// POUs/Diverse/FB_SafetyElementAnz
// Dieser FB dient zur Erweiterung eines älteren Schutztürbausteins für die Anzeige (nur Anzeige keine Fehlermeldung) in der Avalon-HMI im DataCrtlView oder PlcStructure.
// Zudem kann er noch als AnzeigeFB für Lichtgitter oder einzelne Nothalte genuzt werden.
FUNCTION_BLOCK FB_SafetyElementAnz
VAR_IN_OUT
	IQ_stOpVisual			:ST_OP_Visual;	// Zur Anzeige der Schutztür mit Nothalt oder auch Lichtgitter in der HMI
END_VAR
VAR_INPUT
	I_bTuerGeschlossen	: BOOL	:= TRUE;	// Türschalter: TwinSAFE-Kanal 1 geschlossen, oder Lichtgitter OK, oder wenn nur der Nothalt zur Anzeige gebracht wird, weglassen
	I_bTuerGeschlUndVerr	: BOOL	:= TRUE;	// Türschalter: TwinSAFE-Kanal 2 verriegelt, oder Lichtgitter OK, oder wenn nur der Nothalt zur Anzeige gebracht wird, weglassen
	I_bAutoHalt				: BOOL;	// Autohalt der Schutztür aktiv
	I_bNotHalt				: BOOL	:= TRUE;	//	Nothalt an der Schutztür wurde gedrückt, bei Lichtgitter einfach weglassen
	I_bTakt					: BOOL;	//  blinktakt für Q_bAnzeige
	I_sPfadImage			: STRING	:='Objekt-Schiebetuer.svg';	//Pfad für das anzuzeigende Icon
END_VAR
VAR_OUTPUT
	Q_nAnzeige				: DWORD;	// Für die Anzeige im DataCrtlView: Farbe, rot bei Nothalt, gelb bei offen und blau bei Automatik-Halt
	Q_bAnzeige				: BOOL;	// Für die Anzeige im DataCrtlView: TRUE bei Nothalt oder wenn die Tür nicht geschlossen und verriegelt ist
END_VAR

IQ_stOpVisual.sImage := I_sPfadImage;

IF NOT I_bNotHalt
THEN
	IQ_stOpVisual.sColour := cRotAsString;
	IQ_stOpVisual.iDisplayMode := 1;
	Q_bAnzeige	:= TRUE;
	IF I_bTakt
	THEN
		Q_nAnzeige	:= cRot;
	ELSE
		Q_nAnzeige	:= cKEYBACK;
	END_IF
ELSIF I_bTuerGeschlossen
	AND I_bTuerGeschlUndVerr
	AND I_bAutoHalt
THEN
	IQ_stOpVisual.iDisplayMode := 1;
	IQ_stOpVisual.sColour := cBlauAsString;
ELSIF I_bTuerGeschlossen
	AND I_bTuerGeschlUndVerr
THEN
	IQ_stOpVisual.sColour := cDefaultAsString;
	Q_bAnzeige	:= FALSE;
	Q_nAnzeige	:= cKEYBACK;
	IQ_stOpVisual.iDisplayMode := 3;
ELSE
	IQ_stOpVisual.sColour := cGelbAsString;
	IQ_stOpVisual.iDisplayMode := 1;
	Q_bAnzeige	:= TRUE;
	IF I_bTakt
	THEN
		Q_nAnzeige	:= cGelb;
	ELSE
		Q_nAnzeige	:= cKEYBACK;
	END_IF
END_IF

END_FUNCTION_BLOCK

// POUs/Diverse/FB_UsvStatus
// Dieser Baustein wertet die lokale USV aus und beschreibt die Meldungen.
// Es ist eigentlich nur eine Übersetzung von dem USV-Baustein auf die Avalon-Meldungen
FUNCTION_BLOCK FB_UsvStatus
VAR_INPUT
	I_nLevelLowPercent		:	DWORD:= 30;
	I_nLevelCriticalPercent	:	DWORD:= 15;
END_VAR
VAR_IN_OUT
	IQ_stMeldung			: ST_MeldUSV;
END_VAR
VAR
	fbGetUPSStatus		:	Tc2_IoFunctions.FB_GetUPSStatus;
END_VAR

fbGetUPSStatus(
	sNetId		:=	'',
	nPort			:=	0,		// 0 = Windows UPS service
	bEnable		:=	TRUE
);

IQ_stMeldung.bMeldAustausch			:= fbGetUPSStatus.stStatus.eBatteryStatus	=	Tc2_IoFunctions.BatteryReplace;
IQ_stMeldung.bMeldBatteriebetrieb	:= fbGetUPSStatus.stStatus.ePowerStatus	=	Tc2_IoFunctions.PowerOnBattery;
IQ_stMeldung.bMeldKommFehler			:= fbGetUPSStatus.stStatus.eCommStatus	=	Tc2_IoFunctions.UpsCommFailed;
IQ_stMeldung.bMeldKritLevel			:= fbGetUPSStatus.stStatus.BatteryLifePercent < I_nLevelCriticalPercent;
IQ_stMeldung.bMeldStatusUnbekannt	:= fbGetUPSStatus.stStatus.eCommStatus	=	Tc2_IoFunctions.UpsCommUnknownStatus;
IQ_stMeldung.bMeldUnteresLevel		:= fbGetUPSStatus.stStatus.BatteryLifePercent < I_nLevelLowPercent
													AND fbGetUPSStatus.stStatus.ePowerStatus	=	Tc2_IoFunctions.PowerOnBattery;
// ENDE

END_FUNCTION_BLOCK

// POUs/Diverse/FB_WartgTuer
// OBSOLET! Wird nicht weiter supportet. FB für eine Wartungstür. Noch keine Adaption an die Avalon-HMI.
// Es sollte der FB_WartgTuerMeld genutzt werden.
FUNCTION_BLOCK FB_WartgTuer
VAR_INPUT
	I_bFreigTuerEntrieg	:BOOL;	//Allgem. Türfreigabe durch PLC
	I_bAnAbwTastEntrieg	:BOOL;
	I_bQuittTastVerrieg	:BOOL;
	I_bAbfrgTuerGeschl	:BOOL;	//Türschalter: TwinSAFE-Kanal 1
	I_bAbfrgTuerMagnet	:BOOL;	//Türschalter: TwinSAFE-Kanal 2	
	I_bEntrgMeldMagnet	:BOOL;	//Rückmeldung vom Safety-Projekt
	I_bHinwTaktEntrieg	:BOOL;
	I_bHinwTaktEntrglt	:BOOL;

	I_bAutomBetrAngew		:BOOL;
	I_bTastAutomForts		:BOOL;
	I_bUeberbrSteuerhilfsluft	: BOOL;
END_VAR
VAR_OUTPUT

	Q_bAnwTuerEntrieg		:BOOL; 
	Q_bTuerEntriegelt		:BOOL; 
	Q_bAnwQuittMeldg		:BOOL; 
	Q_bEntrgAnfdMagnet	:BOOL;	//Anforderung an Safety-Projekt

	Q_bAutomHaltAktiv		:BOOL;
	Q_bAutomHaltMeldg		:BOOL;	
	
	Q_bAutomHaltMeldgHin	:BOOL;
	
END_VAR
VAR

	
	rtrigAnwQuittTast		:R_TRIG;
	bAnwahlEntriegeln		:BOOL;
	bMagnetEntriegeln		:BOOL;
	bMagnetEntriegelt		:BOOL;
	
	rtrigTastAutoForts	:R_TRIG;
	bAutomHaltManForts	:BOOL;
	
	tonInit					:TON;
	
END_VAR

a_TuerEntrieg ();
b_AutomHalt ();

ACTION a_TuerEntrieg:

//Init, da die Signale aus der Safety nicht sofort da sind und dann die Türen sich öffnen	
tonInit(	IN:= TRUE,
			PT:= T#5S);	
	
IF tonInit.Q
	AND bTwinSAFEInRun
THEN

	rtrigAnwQuittTast (CLK:= I_bAnAbwTastEntrieg
							  		 OR I_bQuittTastVerrieg); 
	
	IF I_bAnAbwTastEntrieg
		AND rtrigAnwQuittTast.Q
		AND NOT bMagnetEntriegelt
	THEN
		bAnwahlEntriegeln:= NOT bAnwahlEntriegeln;	
	END_IF
	
	IF (I_bQuittTastVerrieg
		AND rtrigAnwQuittTast.Q)	
		AND I_bAbfrgTuerGeschl
	THEN
		bMagnetEntriegeln:=	
		bMagnetEntriegelt:= FALSE;	
	END_IF	

	IF (bAnwahlEntriegeln
			AND I_bFreigTuerEntrieg)
		OR NOT I_bAbfrgTuerGeschl
		OR (NOT I_bQuittTastVerrieg
				AND NOT I_bAbfrgTuerMagnet) 
	THEN
		bMagnetEntriegeln:= TRUE;		

		IF I_bEntrgMeldMagnet 
		THEN
			bAnwahlEntriegeln:= FALSE;
			bMagnetEntriegelt:= TRUE;	
		END_IF
   END_IF

	(*Ausgangszuweisung*)

	Q_bAnwTuerEntrieg := bAnwahlEntriegeln;
	
	Q_bTuerEntriegelt	:= bMagnetEntriegelt;
	
	Q_bAnwQuittMeldg	:= (bAnwahlEntriegeln
									AND I_bHinwTaktEntrieg) 
								OR ((NOT I_bAbfrgTuerGeschl
										OR NOT I_bAbfrgTuerMagnet)
									AND I_bHinwTaktEntrglt)
								OR (NOT bAnwahlEntriegeln
										AND NOT bMagnetEntriegeln);	 

	Q_bEntrgAnfdMagnet:= bMagnetEntriegeln;		
END_IF
END_ACTION

ACTION b_AutomHalt:
	(*Abfrage/Quittierung*)

	rtrigTastAutoForts (CLK:= I_bTastAutomForts
										AND NOT I_bAnAbwTastEntrieg );
	
	IF I_bAutomBetrAngew
		AND bMagnetEntriegelt
	THEN
		bAutomHaltManForts:= TRUE;	
	ELSIF rtrigTastAutoForts.Q 
	THEN
			bAutomHaltManForts:= FALSE;	
   END_IF

	(*Ausgangszuweisung*)

	Q_bAutomHaltAktiv	:= bAutomHaltManForts;
	
	Q_bAutomHaltMeldg	:= (NOT bMagnetEntriegelt
									AND bAutomHaltManForts
									AND I_bHinwTaktEntrglt)
								OR (I_bUeberbrSteuerhilfsluft
										AND (bAnwahlEntriegeln
												OR bMagnetEntriegelt)
									AND NOT I_bHinwTaktEntrglt);
								
	Q_bAutomHaltMeldgHin := NOT bMagnetEntriegelt
									AND bAutomHaltManForts;
END_ACTION

END_FUNCTION_BLOCK

// POUs/Diverse/FB_WartgTuerMeld
// FB für eine Wartungstür mit einem Taster zum Umschalten der Schutztüranforderung/Quittierung und einem Taster für Automatikablauf starten.
// Dieser FB ist für die Verwendung mit der Avalon-HMI vorgesehen.
FUNCTION_BLOCK FB_WartgTuerMeld
VAR_IN_OUT		
	IQ_stMeldHMI			:ST_MeldWartgTuer;	// HMI-Strukturen
END_VAR
VAR_INPUT
	I_sName					:STRING;	// Name der Schutztür
	I_sBMK					:STRING;	// z.B.:"ST1020"
	I_bFreigTuerEntrieg	:BOOL;	// Allgem. Türfreigabe durch PLC
	I_bAnAbwTastEntrieg	:BOOL;	// Hardwaretaste für Schutztür anfordern/quittieren
	I_bQuittTastVerrieg	:BOOL;	// Hardwaretaste für Schutztür anfordern/quittieren
	I_bAbfrgTuerGeschl	:BOOL;	// Türschalter: TwinSAFE-Kanal 1
	I_bAbfrgTuerMagnet	:BOOL;	// Türschalter: TwinSAFE-Kanal 2	
	I_bEntrgMeldMagnet	:BOOL;	// Rückmeldung vom Safety-Projekt
	I_bHinwTaktEntrieg	:BOOL;	// mittlerer Takt, ggf. 1Hz
	I_bHinwTaktEntrglt	:BOOL;	// schneller Takt, ggf. 5Hz

	I_bAutomBetrAngew		:BOOL;	// Signal das Automatikablauf angewählt ist.
	I_bTastAutomForts		:BOOL;	// Hardwaretaste für Automatikablauf fortsetzen
	I_bUeberbrSteuerhilfsluft	: BOOL;	// Signal aus dem Safety: Steuerhilfluft ist überbrückt
	
	I_bMeldFreigabe		:BOOL	:= TRUE;	// Hiermit wird die Meldung in der HMI freigegeben. Dieser Eingang kann mit TwinSAFE_OK (oder ähnliches) beschrieben werden, damit die Meldung bei einem Safetyfehler nicht angezeigt werden und unnötig die Meldungen zumüllen.
END_VAR
VAR_OUTPUT

	Q_bAnwTuerEntrieg		:BOOL; 	// Meldung Wartungstür ist zum Entriegeln angwählt
	Q_bTuerEntriegelt		:BOOL;	// Meldung Wartungstür ist entriegelt
	Q_bAnwQuittMeldg		:BOOL;	// Leuchtmelder für den Taster Schutztür anfordern/quittieren
	Q_bEntrgAnfdMagnet	:BOOL;	// Anforderung an Safety-Projekt

	Q_bAutomHaltAktiv		:BOOL;	// Meldung Automatik-Halt ist aktiv
	Q_bAutomHaltMeldg		:BOOL;	// Leuchtmelder für den Taster Automatikablauf fortsetzen
	
	Q_bAutomHaltMeldgHin	:BOOL;	// Meldung das Automatik-Halt noch aktiv ist, obwohl Schutztür geschlossen ist.
	
END_VAR
VAR

	
	rtrigAnwQuittTast		:R_TRIG;
	bAnwahlEntriegeln		:BOOL;
	bMagnetEntriegeln		:BOOL;
	bMagnetEntriegelt		:BOOL;
	
	rtrigTastAutoForts	:R_TRIG;
	bAutomHaltManForts	:BOOL;
	
	tonInit					:TON;
	
END_VAR

a_TuerEntrieg ();
b_AutomHalt ();
z_Meld();

ACTION a_TuerEntrieg:

//Init, da die Signale aus der Safety nicht sofort da sind und dann die Türen sich öffnen	
tonInit(	IN:= TRUE,
			PT:= T#5S);	
	
IF tonInit.Q
	AND bTwinSAFEInRun
THEN

	rtrigAnwQuittTast (CLK:= I_bAnAbwTastEntrieg
							  		 OR I_bQuittTastVerrieg); 
	
	IF I_bAnAbwTastEntrieg
		AND rtrigAnwQuittTast.Q
		AND NOT bMagnetEntriegelt
	THEN
		bAnwahlEntriegeln:= NOT bAnwahlEntriegeln;	
	END_IF
	
	IF (I_bQuittTastVerrieg
		AND rtrigAnwQuittTast.Q)	
		AND I_bAbfrgTuerGeschl
	THEN
		bMagnetEntriegeln:=	
		bMagnetEntriegelt:= FALSE;	
	END_IF	

	IF (bAnwahlEntriegeln
			AND I_bFreigTuerEntrieg)
		OR NOT I_bAbfrgTuerGeschl
		OR (NOT I_bQuittTastVerrieg
				AND NOT I_bAbfrgTuerMagnet) 
	THEN
		bMagnetEntriegeln:= TRUE;		

		IF I_bEntrgMeldMagnet 
		THEN
			bAnwahlEntriegeln:= FALSE;
			bMagnetEntriegelt:= TRUE;	
		END_IF
   END_IF

	(*Ausgangszuweisung*)

	Q_bAnwTuerEntrieg := bAnwahlEntriegeln;
	
	Q_bTuerEntriegelt	:= bMagnetEntriegelt;
	
	Q_bAnwQuittMeldg	:= (bAnwahlEntriegeln
									AND I_bHinwTaktEntrieg) 
								OR ((NOT I_bAbfrgTuerGeschl
										OR NOT I_bAbfrgTuerMagnet)
									AND I_bHinwTaktEntrglt)
								OR (NOT bAnwahlEntriegeln
									AND NOT bMagnetEntriegeln);	 

	Q_bEntrgAnfdMagnet:= bMagnetEntriegeln;		
END_IF
END_ACTION

ACTION b_AutomHalt:
	(*Abfrage/Quittierung*)

	rtrigTastAutoForts (CLK:= I_bTastAutomForts
										AND NOT I_bAnAbwTastEntrieg );
	
	IF I_bAutomBetrAngew
		AND bMagnetEntriegelt
	THEN
		bAutomHaltManForts:= TRUE;	
	ELSIF rtrigTastAutoForts.Q 
	THEN
			bAutomHaltManForts:= FALSE;	
   END_IF

	(*Ausgangszuweisung*)

	Q_bAutomHaltAktiv	:= bAutomHaltManForts;
	
	Q_bAutomHaltMeldg	:= (NOT bMagnetEntriegelt
									AND bAutomHaltManForts
									AND I_bHinwTaktEntrglt)
								OR (I_bUeberbrSteuerhilfsluft
										AND (bAnwahlEntriegeln
												OR bMagnetEntriegelt)
									AND NOT I_bHinwTaktEntrglt);
								
	Q_bAutomHaltMeldgHin := NOT bMagnetEntriegelt
									AND bAutomHaltManForts;
END_ACTION

ACTION z_Meld:


IQ_stMeldHMI.SourceName		 	:= 'Schutztür';
IQ_stMeldHMI.sBMK		 			:= I_sBMK;
IQ_stMeldHMI.sAktorName		 	:= I_sName;
IQ_stMeldHMI.bMeldAutoHalt 	:= Q_bAutomHaltAktiv
											AND NOT Q_bTuerEntriegelt;
											
IQ_stMeldHMI.bMeldGeoeffnet 	:= (NOT I_bAbfrgTuerGeschl
												OR NOT I_bAbfrgTuerMagnet)
											AND I_bMeldFreigabe;
											
IQ_stMeldHMI.bMeldAnwahl		:= bAnwahlEntriegeln
											AND I_bAbfrgTuerMagnet;
END_ACTION

END_FUNCTION_BLOCK

// POUs/Diverse/FB_WartgTuerMeldAnz
// FB für eine Wartungstür mit einem Taster zum Umschalten der Schutztüranforderung/Quittierung und einem Taster für Automatikablauf starten.
// Dieser FB ist für die Verwendung mit der Avalon-HMI vorgesehen und wurde durch eine Anzeigemöglichkeit mit ST_OP_Visual in der Avalon-HMI erweitert.
FUNCTION_BLOCK FB_WartgTuerMeldAnz
VAR_IN_OUT		
	IQ_stMeldHMI			:ST_MeldWartgTuer;	// HMI-Strukturen
	IQ_stOpVisual			:ST_OP_Visual;	// Zur Anzeige der Schutztür mit Nothalt in der HMI
END_VAR
VAR_INPUT
	I_sName					:STRING;	// Name der Schutztür
	I_sBMK					:STRING;	// z.B.:"ST1020"
	I_bFreigTuerEntrieg	:BOOL;	// Allgem. Türfreigabe durch PLC
	I_bAnAbwTastEntrieg	:BOOL;	// Hardwaretaste für Schutztür anfordern/quittieren
	I_bQuittTastVerrieg	:BOOL;	// Hardwaretaste für Schutztür anfordern/quittieren
	I_bAbfrgTuerGeschl	:BOOL;	// Türschalter: TwinSAFE-Kanal 1
	I_bAbfrgTuerMagnet	:BOOL;	// Türschalter: TwinSAFE-Kanal 2	
	I_bEntrgMeldMagnet	:BOOL;	// Rückmeldung vom Safety-Projekt
	I_bHinwTaktEntrieg	:BOOL;	// mittlerer Takt, ggf. 1Hz
	I_bHinwTaktEntrglt	:BOOL;	// schneller Takt, ggf. 5Hz
	
	I_bAutomBetrAngew		:BOOL;	// Signal das Automatikablauf angewählt ist.
	I_bTastAutomForts		:BOOL;	// Hardwaretaste für Automatikablauf fortsetzen
	I_bUeberbrSteuerhilfsluft	: BOOL;	// Signal aus dem Safety: Steuerhilfluft ist überbrückt
	
	I_bMeldFreigabe		:BOOL	:= TRUE;	// Hiermit wird die Meldung in der HMI freigegeben. Dieser Eingang kann mit TwinSAFE_OK (oder ähnliches) beschrieben werden, damit die Meldung bei einem Safetyfehler nicht angezeigt werden und unnötig die Meldungen zumüllen.
	I_sPfadImage			:STRING	:='Objekt-Schiebetuer.svg';			//Pfad für das anzuzeigende Icon
	I_bNotHalt				:BOOL	:= TRUE;	// Not-Halt an dieser Tür wurde gedrückt. Kann weggelassen werden. Blink dann aber nicht rot
END_VAR
VAR_OUTPUT

	Q_bAnwTuerEntrieg		:BOOL; 	// Meldung Wartungstür ist zum Entriegeln angwählt
	Q_bTuerEntriegelt		:BOOL;	// Meldung Wartungstür ist entriegelt
	Q_bAnwQuittMeldg		:BOOL;	// Leuchtmelder für den Taster Schutztür anfordern/quittieren
	Q_bEntrgAnfdMagnet	:BOOL;	// Anforderung an Safety-Projekt

	Q_bAutomHaltAktiv		:BOOL;	// Meldung Automatik-Halt ist aktiv
	Q_bAutomHaltMeldg		:BOOL;	// Leuchtmelder für den Taster Automatikablauf fortsetzen
	
	Q_bAutomHaltMeldgHin	:BOOL;	// Meldung das Automatik-Halt noch aktiv ist, obwohl Schutztür geschlossen ist.
	
	Q_nAnzeige				: DWORD;	// Für die Anzeige im DataCrtlView: Farbe, rot bei Nothalt, gelb bei offen und blau bei Automatik-Halt
	Q_bAnzeige				: BOOL;	// Für die Anzeige im DataCrtlView: TRUE bei Nothalt oder wenn die Tür nicht geschlossen und verriegelt ist
	
END_VAR
VAR

	
	rtrigAnwQuittTast		:R_TRIG;
	bAnwahlEntriegeln		:BOOL;
	bMagnetEntriegeln		:BOOL;
	bMagnetEntriegelt		:BOOL;
	
	rtrigTastAutoForts	:R_TRIG;
	bAutomHaltManForts	:BOOL;
	
	tonInit					:TON;
	
END_VAR

a_TuerEntrieg ();
b_AutomHalt ();
c_Anzeige();
z_Meld();

ACTION a_TuerEntrieg:

//Init, da die Signale aus der Safety nicht sofort da sind und dann die Türen sich öffnen	
tonInit(	IN:= TRUE,
			PT:= T#5S);	
	
IF tonInit.Q
	AND bTwinSAFEInRun
THEN

	rtrigAnwQuittTast (CLK:= I_bAnAbwTastEntrieg
							  		 OR I_bQuittTastVerrieg); 
	
	IF I_bAnAbwTastEntrieg
		AND rtrigAnwQuittTast.Q
		AND NOT bMagnetEntriegelt
	THEN
		bAnwahlEntriegeln:= NOT bAnwahlEntriegeln;	
	END_IF
	
	IF (I_bQuittTastVerrieg
		AND rtrigAnwQuittTast.Q)	
		AND I_bAbfrgTuerGeschl
	THEN
		bMagnetEntriegeln:=	
		bMagnetEntriegelt:= FALSE;	
	END_IF	

	IF (bAnwahlEntriegeln
			AND I_bFreigTuerEntrieg)
		OR NOT I_bAbfrgTuerGeschl
		OR (NOT I_bQuittTastVerrieg
				AND NOT I_bAbfrgTuerMagnet) 
	THEN
		bMagnetEntriegeln:= TRUE;		

		IF I_bEntrgMeldMagnet 
		THEN
			bAnwahlEntriegeln:= FALSE;
			bMagnetEntriegelt:= TRUE;	
		END_IF
   END_IF

	(*Ausgangszuweisung*)

	Q_bAnwTuerEntrieg := bAnwahlEntriegeln;
	
	Q_bTuerEntriegelt	:= bMagnetEntriegelt;
	
	Q_bAnwQuittMeldg	:= (bAnwahlEntriegeln
									AND I_bHinwTaktEntrieg) 
								OR ((NOT I_bAbfrgTuerGeschl
										OR NOT I_bAbfrgTuerMagnet)
									AND I_bHinwTaktEntrglt)
								OR (NOT bAnwahlEntriegeln
									AND NOT bMagnetEntriegeln);	 

	Q_bEntrgAnfdMagnet:= bMagnetEntriegeln;		
END_IF
END_ACTION

ACTION b_AutomHalt:
	(*Abfrage/Quittierung*)

	rtrigTastAutoForts (CLK:= I_bTastAutomForts
										AND NOT I_bAnAbwTastEntrieg );
	
	IF I_bAutomBetrAngew
		AND bMagnetEntriegelt
	THEN
		bAutomHaltManForts:= TRUE;	
	ELSIF rtrigTastAutoForts.Q 
	THEN
			bAutomHaltManForts:= FALSE;	
   END_IF

	(*Ausgangszuweisung*)

	Q_bAutomHaltAktiv	:= bAutomHaltManForts;
	
	Q_bAutomHaltMeldg	:= (NOT bMagnetEntriegelt
									AND bAutomHaltManForts
									AND I_bHinwTaktEntrglt)
								OR (I_bUeberbrSteuerhilfsluft
										AND (bAnwahlEntriegeln
												OR bMagnetEntriegelt)
									AND NOT I_bHinwTaktEntrglt);
								
	Q_bAutomHaltMeldgHin := NOT bMagnetEntriegelt
									AND bAutomHaltManForts;
END_ACTION

ACTION c_Anzeige:
IQ_stOpVisual.sImage := I_sPfadImage;

IF NOT I_bNotHalt
THEN
	IQ_stOpVisual.sColour := cRotAsString;
	IQ_stOpVisual.iDisplayMode := 1;
	Q_bAnzeige	:= TRUE;
	IF bTaktMittel
	THEN
		Q_nAnzeige	:= cRot;
	ELSE
		Q_nAnzeige	:= cKEYBACK;
	END_IF
ELSIF I_bAbfrgTuerGeschl
	AND I_bAbfrgTuerMagnet
	AND bAutomHaltManForts
THEN
	IQ_stOpVisual.iDisplayMode := 1;
	IQ_stOpVisual.sColour 		:= cBlauAsString;
	Q_bAnzeige						:= TRUE;
	IF bTaktMittel
	THEN
		Q_nAnzeige	:= cBlau;
	ELSE
		Q_nAnzeige	:= cKEYBACK;
	END_IF
ELSIF I_bAbfrgTuerGeschl
	AND I_bAbfrgTuerMagnet
THEN
	IQ_stOpVisual.sColour := cDefaultAsString;
	Q_bAnzeige	:= FALSE;
	Q_nAnzeige	:= cKEYBACK;
	IQ_stOpVisual.iDisplayMode := 3;
ELSE
	IQ_stOpVisual.sColour := cGelbAsString;
	IQ_stOpVisual.iDisplayMode := 1;
	Q_bAnzeige	:= TRUE;
	IF bTaktMittel
	THEN
		Q_nAnzeige	:= cGelb;
	ELSE
		Q_nAnzeige	:= cKEYBACK;
	END_IF
END_IF
END_ACTION

ACTION z_Meld:


IQ_stMeldHMI.SourceName		 	:= 'Schutztür';
IQ_stMeldHMI.sBMK		 			:= I_sBMK;
IQ_stMeldHMI.sAktorName		 	:= I_sName;
IQ_stMeldHMI.bMeldAutoHalt 	:= Q_bAutomHaltAktiv
											AND NOT Q_bTuerEntriegelt;
											
IQ_stMeldHMI.bMeldGeoeffnet 	:= (NOT I_bAbfrgTuerGeschl
												OR NOT I_bAbfrgTuerMagnet)
											AND I_bMeldFreigabe;
											
IQ_stMeldHMI.bMeldAnwahl		:= bAnwahlEntriegeln
											AND I_bAbfrgTuerMagnet;
END_ACTION

END_FUNCTION_BLOCK

// POUs/EAP/FB_EAP_Kommunikation
FUNCTION_BLOCK FB_EAP_Kommunikation
VAR CONSTANT
	nMaxFehlerCounter						: INT := 3;
END_VAR
VAR_INPUT
	I_sNamePartner						: STRING;					// Klartextname der Partneranlage
	I_nFortlaufendeID					: INT;						// Fortlaufende ID
	I_bOhneTwinSAFE					: BOOL;						// Deaktiviert die TwinSAFE Überprüfung und Abarbeitung
	
 	I_nKommBits								: DWORD;					// Kommunikations-Bits aus dem PLC Programm heraus
	I_stTwinSAFEGroupInfoData			: ST_TwinSAFE_Group_Info;	// InfoData der TwinSAFE Gruppe fals TwinSAFE vorhanden
	I_stTwinSAFEConnectionInfoData	: ST_TwinSAFEConnInfo4Byte;// InfoData der TwinSAFE Connection falls vorhanden
	I_bFehlerEtherCAT						: BOOL;						// "glb_bFehler_EtherCATAllg"
	I_bSafetyFreigabe						: BOOL;						// "glb_bSafetyFrg"
	
	I_tSendeTaktZeit						: TIME := t#250ms;
	
	{attribute 'hide' := ''}
	I_bDeaktivieren						: BOOL;						// Deaktiviert die Kommunikation sowie die Auswertung
	{attribute 'hide' := ''}
	I_bReset									: BOOL;						// Reset für z.B. anstehende Meldungen
END_VAR
VAR_IN_OUT
	{attribute 'hide' := ''}
	IQ_EAP_Partner_Empfangen			: ST_EAP_Receive;
	{attribute 'hide' := ''}
	IQ_EAP_Partner_Senden				: ST_EAP_Send;
END_VAR
VAR_OUTPUT
	Q_bFehler								: BOOL; 		//Quittierungspflichtiger Fehler liegt an
	Q_bSendeBereit							: BOOL;		// Baustein ist bereit einen neuen Datensatz zu senden
	Q_bNeueDaten							: BOOL;		// Neue Daten von Partner sind vorhanden und können abgerufen werden
	Q_bTwinSAFEReset						: BOOL;		// Quittierungsausgang für zugehörige TwinSAFE Gruppe
	Q_nKommBits								: DWORD;		// Komminkationsbits mit Partneranlage
	Q_bPartnerLebt							: BOOL;		// Verbindung uzm Partner steht
	Q_stTwinSAFEConnection				: ST_TwinSAFE_Connection;
	Q_stMeld									: ST_MeldEAPKommError;
													(*	 1 = schlechte Qualität
														 2 = Keine Kommunikation
														 3 = Falsche ID zurückgemeldet
														 4 = TwinSAFE Gruppe in STörung
														 5 = Unbekannter TwinSAFE Fehler
														 6 = TwinSAFE Connection im ungültigen Zustand
														 7 = 
														 8 = 
														 9 = 
														 10 = 
													*)	
END_VAR
VAR
	bInit									: BOOL;
	arrDatenBuffer						: ARRAY[1..10] OF ST_TempEAPDaten;
	bPartnerLebt						: BOOL;
	
	tonTimeOut,
	tonWaitSend,
	tonWaitReceive						: TON;
	
	nStepBereit,
	nFehlerCounter,
	nIndx									: INT;

	stStepSend,
	stStepReceive			        	: ST_StepCtrl;

	bGrpReset							: BOOL;
	tpReset								: TP;
	nLastCycleIndex,
	nLastCycleTOut						: UINT;
	
	stTempDatenSend					: ST_TempEAPDaten;
	
	nOldTwinSAFEGroupMapState,
	nOldTwinSAFEConnectionMapState		: USINT;
	
	rtrigDeaktiviert					: R_TRIG;
	
	bInvalidFramestate				: BOOL;

END_VAR

IF NOT bInit THEN
	_00_Init();
ELSE
	
	rtrigDeaktiviert(CLK := I_bDeaktivieren);
	
	tonTimeOut(IN:= NOT tonTimeOut.Q, PT := I_tSendeTaktZeit);
	
	IF tonTimeOut.Q
	AND NOT I_bDeaktivieren
	THEN
		Q_bPartnerLebt	:=
		bPartnerLebt 	:= 
			(IQ_EAP_Partner_Empfangen.CycleIndex 
				<> nLastCycleTOut)
			AND (IQ_EAP_Partner_Empfangen.Quality 
				< 4000);
		
		Q_stMeld.bMeldKommError := 
			(	IQ_EAP_Partner_Empfangen.CycleIndex 
				= nLastCycleTOut);
		
		Q_stMeld.bMeldKeinSignal := 
			IQ_EAP_Partner_Empfangen.Quality 
			> 4000 // Wert erstmal testweise, bei langen Leitungen prüfen ob erhöht werden muss 
			AND NOT Q_stMeld.bMeldKommError;
																
		nLastCycleTOut := IQ_EAP_Partner_Empfangen.CycleIndex;
	END_IF
	
	IF (I_bReset
		AND Q_bFehler)
	OR rtrigDeaktiviert.Q
	THEN
		IQ_EAP_Partner_Senden.VarData.Data.KommBits		:= 0;
		Q_nKommBits													:= 0;

		stStepSend.IQ.nStep										:= 0;
		stStepReceive.IQ.nStep									:= 0;

		nStepBereit													:= 0;
		bPartnerLebt												:= 0;

		MEMSET(ADR(IQ_EAP_Partner_Senden.VarData), 0, SIZEOF(IQ_EAP_Partner_Senden.VarData));
		IQ_EAP_Partner_Senden.VarData.Data.TeilID			:= '0';
		MEMSET(ADR(stTempDatenSend), 0, SIZEOF(stTempDatenSend));
		
		Q_stMeld.bMeldKommError			:=
		Q_stMeld.bMeldKeinSignal			:=
		Q_stMeld.bMeldFalscheID			:=
		Q_stMeld.bMeldTwinSafeGrp			:=
		Q_stMeld.bMeldTwinSafeFehler		:=
		Q_stMeld.bMeldTwinSafeUngueltig	:= FALSE;
	END_IF
	
	IF NOT I_bDeaktivieren 
	THEN
		IQ_EAP_Partner_Senden.VarCtrl		 				:= 0;
		IQ_EAP_Partner_Senden.VarData.Data.KommBits	:= I_nKommBits;
		
		IF bPartnerLebt
		THEN
			Q_nKommBits		:= IQ_EAP_Partner_Empfangen.VarData.Data.KommBits;
			m_Send();
			m_Receive();	
		ELSE
			Q_bSendeBereit := FALSE;
		END_IF
	
	ELSE	
		IQ_EAP_Partner_Senden.VarCtrl		 				:= 1;
		IQ_EAP_Partner_Senden.VarData.Data.KommBits	:= 0;
		Q_nKommBits		:= 0;
	END_IF
	
	CASE nStepBereit OF
		0: // auf neue Daten prüfen
			Q_bNeueDaten	:= FALSE;
			IF   arrDatenBuffer[1].sTeilenummer <> '' 
			 AND arrDatenBuffer[1].sTeilenummer <> '0'
			THEN
				nStepBereit	:= 5;
			END_IF
	
		5: // Setzen des "Neue Daten" bits
			Q_bNeueDaten	:= TRUE;
			nStepBereit		:= 10;
			
		10: //Warteschritt
			;
			
		15:// Rücksprung
			nStepBereit		:= 0;
	
	END_CASE
	
	Q_bFehler 	:= Q_stMeld.bMeldFalscheID;
	
	IF NOT I_bOhneTwinSAFE
	THEN
		_02_TwinSAFE();
	END_IF

END_IF

ACTION _00_Init:

	Q_stMeld.sAnlagenteil	:= I_sNamePartner;

	bInit := TRUE;
END_ACTION

ACTION _02_TwinSAFE:

IF tonTimeOut.Q
AND NOT I_bFehlerEtherCAT
AND I_bSafetyFreigabe
THEN

	CASE I_stTwinSAFEGroupInfoData.nMapState OF
		1: 
			bGrpReset						:= 
			Q_bTwinSAFEReset				:= 
			Q_stMeld.bMeldTwinSafeGrp		:=
			Q_stMeld.bMeldTwinSafeFehler	:= FALSE;
	
		2..5:
			bGrpReset						:= NOT bGrpReset;
			Q_stMeld.bMeldTwinSafeGrp		:= TRUE;
			
		ELSE
			Q_stMeld.bMeldTwinSafeFehler	:= TRUE;
	END_CASE

(*	// Auswertung Gruppe und Reset
	IF (I_stTwinSAFEGroupInfoData.nMapState
		<> nOldTwinSAFEGroupMapState)
	THEN
		nOldTwinSAFEGroupMapState := I_stTwinSAFEGroupInfoData.nMapState;
		
		CASE I_stTwinSAFEGroupInfoData.nMapState OF
			1: 
				bGrpReset						:= FALSE;
				Q_bTwinSAFEReset				:= FALSE;
				fbMeldung[5].I_bAktiv		:= FALSE;
				fbMeldung[4].I_bAktiv		:= FALSE;	
		
			2..5:
				bGrpReset						:= NOT bGrpReset;
				fbMeldung[4].I_bAktiv		:= TRUE;
				
			ELSE
				fbMeldung[5].I_bAktiv		:= TRUE;
		END_CASE
	END_IF
*)	
	// Auswertung der Connection Info
	IF I_stTwinSAFEConnectionInfoData.nMapState
		<> nOldTwinSAFEConnectionMapState
	THEN
		nOldTwinSAFEConnectionMapState := I_stTwinSAFEConnectionInfoData.nMapState;
		CASE I_stTwinSAFEConnectionInfoData.nMapState OF
			104:	
				Q_stMeld.bMeldTwinSafeUngueltig	:= FALSE;
			ELSE
				Q_stMeld.bMeldTwinSafeUngueltig	:= TRUE;
		END_CASE
	END_IF
END_IF

tpReset(IN := bGrpReset, PT := T#250MS, Q=> Q_bTwinSAFEReset);

Q_stTwinSAFEConnection.Q_bIn0 	:= I_stTwinSAFEConnectionInfoData.nInput.0;
Q_stTwinSAFEConnection.Q_bIn1 	:= I_stTwinSAFEConnectionInfoData.nInput.1;
Q_stTwinSAFEConnection.Q_bIn2 	:= I_stTwinSAFEConnectionInfoData.nInput.2;
Q_stTwinSAFEConnection.Q_bIn3 	:= I_stTwinSAFEConnectionInfoData.nInput.3;
Q_stTwinSAFEConnection.Q_bIn4 	:= I_stTwinSAFEConnectionInfoData.nInput.4;
Q_stTwinSAFEConnection.Q_bIn5 	:= I_stTwinSAFEConnectionInfoData.nInput.5;
Q_stTwinSAFEConnection.Q_bIn6 	:= I_stTwinSAFEConnectionInfoData.nInput.6;
Q_stTwinSAFEConnection.Q_bIn7 	:= I_stTwinSAFEConnectionInfoData.nInput.7;

Q_stTwinSAFEConnection.Q_bOut0 	:= I_stTwinSAFEConnectionInfoData.nOutput.0 AND NOT I_bFehlerEtherCAT;
Q_stTwinSAFEConnection.Q_bOut1 	:= I_stTwinSAFEConnectionInfoData.nOutput.1 AND NOT I_bFehlerEtherCAT;
Q_stTwinSAFEConnection.Q_bOut2 	:= I_stTwinSAFEConnectionInfoData.nOutput.2 AND NOT I_bFehlerEtherCAT;
Q_stTwinSAFEConnection.Q_bOut3 	:= I_stTwinSAFEConnectionInfoData.nOutput.3 AND NOT I_bFehlerEtherCAT;
Q_stTwinSAFEConnection.Q_bOut4 	:= I_stTwinSAFEConnectionInfoData.nOutput.4 AND NOT I_bFehlerEtherCAT;
Q_stTwinSAFEConnection.Q_bOut5 	:= I_stTwinSAFEConnectionInfoData.nOutput.5 AND NOT I_bFehlerEtherCAT;
Q_stTwinSAFEConnection.Q_bOut6 	:= I_stTwinSAFEConnectionInfoData.nOutput.6 AND NOT I_bFehlerEtherCAT;
Q_stTwinSAFEConnection.Q_bOut7 	:= I_stTwinSAFEConnectionInfoData.nOutput.7 AND NOT I_bFehlerEtherCAT;
END_ACTION

METHOD PUBLIC m_DatenBereitstellen : ST_TempEAPDaten
VAR_INPUT
END_VAR

IF nStepBereit = 10
THEN
	m_DatenBereitstellen := arrDatenBuffer[1];

	MEMMOVE(ADR(arrDatenBuffer[1]),ADR(arrDatenBuffer[2]),(SIZEOF(arrDatenBuffer)-SIZEOF(arrDatenBuffer[1])));
	MEMSET(ADR(arrDatenBuffer[10]), 0, SIZEOF(arrDatenBuffer[10]));
	nStepBereit		:= 15;
	Q_bNeueDaten	:= FALSE;

ELSE
	m_DatenBereitstellen.sTeilenummer := '0';
END_IF
END_METHOD

METHOD PRIVATE m_Receive : BOOL
VAR_INPUT
END_VAR
{warning disable C0371}
CASE stStepReceive.IQ.nStep OF //		nStepReceive OF
	0:	stStepReceive.IQ.sStatus := 'Warten auf Teile ID';
		tonWaitReceive(
			IN := (		 IQ_EAP_Partner_Empfangen.VarData.Data.TeilID <> '0')
						AND(IQ_EAP_Partner_Empfangen.VarData.Data.TeilID <> '')
						AND(IQ_EAP_Partner_Empfangen.VarData.Data.TeilID <>
							 IQ_EAP_Partner_Senden.VarData.Data.TeilID), 
				PT := T#50MS);
		
		IF tonWaitReceive.Q
		THEN
			tonWaitReceive(IN:=FALSE);
			stStepReceive.IQ.nStep := 5;
		END_IF
		
	5:stStepReceive.IQ.sStatus := 'Kontrolle Zyklus beim Empfangen!';
		IF IQ_EAP_Partner_Empfangen.CycleIndex <> nLastCycleIndex
		AND bPartnerLebt	
		THEN
			nLastCycleIndex 	:= IQ_EAP_Partner_Empfangen.CycleIndex;
			stStepReceive.IQ.nStep := 10;
		ELSE
			;//TODO
		END_IF
		
	10:stStepReceive.IQ.sStatus := 'TeileID: ';
		stStepReceive.IQ.sStatus := CONCAT(stStepReceive.IQ.sStatus, IQ_EAP_Partner_Empfangen.VarData.Data.TeilID);
		stStepReceive.IQ.sStatus := CONCAT(stStepReceive.IQ.sStatus, ' Status: ');
		stStepReceive.IQ.sStatus := CONCAT(stStepReceive.IQ.sStatus, DWORD_TO_STRING(IQ_EAP_Partner_Empfangen.VarData.Data.TeilStatus));
	
		IQ_EAP_Partner_Senden.VarData.Data.TeilID	:= IQ_EAP_Partner_Empfangen.VarData.Data.TeilID;
		
		FOR nIndx := 1 TO 10 BY 1 DO
			IF arrDatenBuffer[nIndx].sTeilenummer = '' 
			THEN 
				arrDatenBuffer[nIndx].sTeilenummer		:= IQ_EAP_Partner_Empfangen.VarData.Data.TeilID;
				arrDatenBuffer[nIndx].wStatus 			:= IQ_EAP_Partner_Empfangen.VarData.Data.TeilStatus;
				arrDatenBuffer[nIndx].wZusatzinfo1		:= IQ_EAP_Partner_Empfangen.VarData.Data.ZusatzInfo1;
				arrDatenBuffer[nIndx].wZusatzinfo2		:= IQ_EAP_Partner_Empfangen.VarData.Data.ZusatzInfo2;
				arrDatenBuffer[nIndx].wZusatzinfo3		:= IQ_EAP_Partner_Empfangen.VarData.Data.ZusatzInfo3;
				arrDatenBuffer[nIndx].wZusatzinfo4		:= IQ_EAP_Partner_Empfangen.VarData.Data.ZusatzInfo4;
				arrDatenBuffer[nIndx].wZusatzinfo5		:= IQ_EAP_Partner_Empfangen.VarData.Data.ZusatzInfo5;
				arrDatenBuffer[nIndx].wZusatzinfo6		:= IQ_EAP_Partner_Empfangen.VarData.Data.ZusatzInfo6;
				arrDatenBuffer[nIndx].wZusatzinfo7		:= IQ_EAP_Partner_Empfangen.VarData.Data.ZusatzInfo7;
				arrDatenBuffer[nIndx].wZusatzinfo8		:= IQ_EAP_Partner_Empfangen.VarData.Data.ZusatzInfo8;
				arrDatenBuffer[nIndx].wZusatzinfo9		:= IQ_EAP_Partner_Empfangen.VarData.Data.ZusatzInfo9;
				arrDatenBuffer[nIndx].wZusatzinfo10		:= IQ_EAP_Partner_Empfangen.VarData.Data.ZusatzInfo10;
				EXIT;
			END_IF
		END_FOR
		stStepReceive.IQ.nStep								:= 15;
		
	15:stStepReceive.IQ.sStatus := 'Warten aus Teile ID gelöscht!';
		IF IQ_EAP_Partner_Empfangen.VarData.Data.TeilID = '0'
		THEN
			stStepReceive.IQ.nStep							:= 20;
		END_IF
		
	20:stStepReceive.IQ.sStatus := 'Kontrolle Zyklus Empfangen Ende!';
		IF IQ_EAP_Partner_Empfangen.CycleIndex <> nLastCycleIndex
		AND bPartnerLebt	
		THEN
			IQ_EAP_Partner_Senden.VarData.Data.TeilID	:= '0';
			nLastCycleIndex 									:= IQ_EAP_Partner_Empfangen.CycleIndex;
			stStepReceive.IQ.nStep							:= 0;
		END_IF
END_CASE
stStepReceive.fbHistory(IQ_StepPara:= stStepReceive.IQ);
END_METHOD

METHOD PRIVATE m_Send : BOOL
VAR_INPUT
END_VAR
{warning disable C0371}
CASE stStepSend.IQ.nStep of  //nStepSend OF
	0:	stStepSend.IQ.sStatus 		:= 'Sendebereit!';
		Q_bSendeBereit 				:= bPartnerLebt;
		                           
	5:	stStepSend.IQ.sStatus 		:= 'Start Senden';
		Q_bSendeBereit 				:= FALSE;
		IF tonTimeOut.Q            
		THEN                       
			stStepSend.IQ.nStep 		:= 10;
		END_IF
		
	10:	stStepSend.IQ.sStatus := 'Kontrolle Sende bereit!';
		IF IQ_EAP_Partner_Senden.FrameState = 0
		THEN
			Q_stMeld.bMeldKeinSignal	:= FALSE;
			nFehlerCounter				:= 0;
			stStepSend.IQ.nStep 		:= 15;
		ELSE
			nFehlerCounter 			:= nFehlerCounter + 1;
			IF nFehlerCounter > nMaxFehlerCounter
			THEN
				Q_stMeld.bMeldKeinSignal	:= TRUE;
				stStepSend.IQ.nStep 		:= 5;
			END_IF
		END_IF
		
	15:	stStepSend.IQ.sStatus := 'Daten in Sendebuffer schreiben! RmNr: ';
		stStepSend.IQ.sStatus := CONCAT( stStepSend.IQ.sStatus,stTempDatenSend.sTeilenummer);
		stStepSend.IQ.sStatus := CONCAT( stStepSend.IQ.sStatus,' Status: ');
		stStepSend.IQ.sStatus := CONCAT( stStepSend.IQ.sStatus,DWORD_TO_STRING(stTempDatenSend.wStatus));
 
		IQ_EAP_Partner_Senden.VarData.Data.TeilID				:= stTempDatenSend.sTeilenummer;
		IQ_EAP_Partner_Senden.VarData.Data.TeilStatus		:= stTempDatenSend.wStatus;
		IQ_EAP_Partner_Senden.VarData.Data.ZusatzInfo1		:= stTempDatenSend.wZusatzinfo1;
		IQ_EAP_Partner_Senden.VarData.Data.ZusatzInfo2		:= stTempDatenSend.wZusatzinfo2;
		IQ_EAP_Partner_Senden.VarData.Data.ZusatzInfo3		:= stTempDatenSend.wZusatzinfo3;
		IQ_EAP_Partner_Senden.VarData.Data.ZusatzInfo4		:= stTempDatenSend.wZusatzinfo4;
		IQ_EAP_Partner_Senden.VarData.Data.ZusatzInfo5		:= stTempDatenSend.wZusatzinfo5;
		IQ_EAP_Partner_Senden.VarData.Data.ZusatzInfo6		:= stTempDatenSend.wZusatzinfo6;
		IQ_EAP_Partner_Senden.VarData.Data.ZusatzInfo7		:= stTempDatenSend.wZusatzinfo7;
		IQ_EAP_Partner_Senden.VarData.Data.ZusatzInfo8		:= stTempDatenSend.wZusatzinfo8;
		IQ_EAP_Partner_Senden.VarData.Data.ZusatzInfo9		:= stTempDatenSend.wZusatzinfo9;
		IQ_EAP_Partner_Senden.VarData.Data.ZusatzInfo10		:= stTempDatenSend.wZusatzinfo10;
		
		stStepSend.IQ.nStep 					:= 20;
		
	20:	stStepSend.IQ.sStatus 					:= 'Zeitverzögerung Senden';
		IF tonTimeOut.Q
		THEN
			stStepSend.IQ.nStep 				:= 25;
		END_IF
		
	25:stStepSend.IQ.sStatus := 'Kontrolle FrameStaus vorm Senden!';
		IF IQ_EAP_Partner_Senden.FrameState = 0
		THEN
			tonWaitSend(IN := FALSE);
			stStepSend.IQ.nStep					:= 30;
		ELSE
			nFehlerCounter 						:= nFehlerCounter +1;
			Q_stMeld.bMeldKeinSignal 				:= TRUE;
			stStepSend.IQ.nStep 					:= 5;
		END_IF
	
	30:	stStepSend.IQ.sStatus 					:= 'Check Vergleich Senden und Rückmeldung RmNr Senden: ';
		stStepSend.IQ.sStatus := CONCAT( stStepSend.IQ.sStatus,IQ_EAP_Partner_Senden.VarData.Data.TeilID) ; 
		stStepSend.IQ.sStatus := CONCAT( stStepSend.IQ.sStatus,' RmNr Empfangen: ') ; 
		stStepSend.IQ.sStatus := CONCAT( stStepSend.IQ.sStatus,IQ_EAP_Partner_Empfangen.VarData.Data.TeilID) ; 
		tonWaitSend(IN := TRUE, PT := T#2S);
		
		IF IQ_EAP_Partner_Empfangen.VarData.Data.TeilID =
			IQ_EAP_Partner_Senden.VarData.Data.TeilID
		AND IQ_EAP_Partner_Empfangen.VarData.Data.TeilID <> '0'	
		THEN  
			IQ_EAP_Partner_Senden.VarData.Data.TeilID			:= '0';
			IQ_EAP_Partner_Senden.VarData.Data.TeilStatus	:= 0;
			IQ_EAP_Partner_Senden.VarData.Data.ZusatzInfo1	:= 0;
			IQ_EAP_Partner_Senden.VarData.Data.ZusatzInfo2	:= 0;
			IQ_EAP_Partner_Senden.VarData.Data.ZusatzInfo3	:= 0;
			IQ_EAP_Partner_Senden.VarData.Data.ZusatzInfo4	:= 0;
			IQ_EAP_Partner_Senden.VarData.Data.ZusatzInfo5	:= 0;
			IQ_EAP_Partner_Senden.VarData.Data.ZusatzInfo6	:= 0;
			IQ_EAP_Partner_Senden.VarData.Data.ZusatzInfo7	:= 0;
			IQ_EAP_Partner_Senden.VarData.Data.ZusatzInfo8	:= 0;
			IQ_EAP_Partner_Senden.VarData.Data.ZusatzInfo9	:= 0;
			IQ_EAP_Partner_Senden.VarData.Data.ZusatzInfo10	:= 0;
			MEMSET(ADR(stTempDatenSend),0,SIZEOF(stTempDatenSend));
			tonWaitSend(IN:=FALSE);
			stStepSend.IQ.nStep 							:= 35;
			
		ELSIF tonWaitSend.Q
		THEN
			tonWaitSend(IN:=FALSE);
			Q_stMeld.sErrorID			:= CONCAT('Gesendete ID: ', IQ_EAP_Partner_Senden.VarData.Data.TeilID); 
			stStepSend.IQ.sStatus 	:= CONCAT( stStepSend.IQ.sStatus,'Fehler beim Senden Gesendete ID: ') ; 
			stStepSend.IQ.sStatus 	:= CONCAT( stStepSend.IQ.sStatus,IQ_EAP_Partner_Senden.VarData.Data.TeilID) ; 
			stStepSend.IQ.nStep 		:= -30;
		END_IF
		
	35: 
		IF tonTimeOut.Q
		THEN
			stStepSend.IQ.nStep 		:= 40;
		END_IF
		
	40:	stStepSend.IQ.sStatus 	:= 'Kontrolle FrameStaus nach dem Senden!';
		IF IQ_EAP_Partner_Senden.FrameState = 0
		THEN
			stStepSend.IQ.nStep		:= 0;
		ELSE
			bInvalidFramestate		:= TRUE;
			stStepSend.IQ.nStep		:= -30;
		END_IF
		
	-30:stStepSend.IQ.sStatus 					:= 'Fehler beim Senden!';
		Q_stMeld.bMeldFalscheID		:= TRUE;
		IF I_bReset
		THEN
			bInvalidFramestate		:= FALSE;
			Q_stMeld.bMeldFalscheID	:= FALSE;
			
			IQ_EAP_Partner_Senden.VarData.Data.TeilID			:= '0';
			IQ_EAP_Partner_Senden.VarData.Data.TeilStatus	:= 0;
			IQ_EAP_Partner_Senden.VarData.Data.ZusatzInfo1	:= 0;
			IQ_EAP_Partner_Senden.VarData.Data.ZusatzInfo2	:= 0;
			IQ_EAP_Partner_Senden.VarData.Data.ZusatzInfo3	:= 0;
			IQ_EAP_Partner_Senden.VarData.Data.ZusatzInfo4	:= 0;
			IQ_EAP_Partner_Senden.VarData.Data.ZusatzInfo5	:= 0;
			IQ_EAP_Partner_Senden.VarData.Data.ZusatzInfo6	:= 0;
			IQ_EAP_Partner_Senden.VarData.Data.ZusatzInfo7	:= 0;
			IQ_EAP_Partner_Senden.VarData.Data.ZusatzInfo8	:= 0;
			IQ_EAP_Partner_Senden.VarData.Data.ZusatzInfo9	:= 0;
			IQ_EAP_Partner_Senden.VarData.Data.ZusatzInfo10	:= 0;
			stStepSend.IQ.nStep 										:= 0;
		END_IF
		
END_CASE
stStepSend.fbHistory(IQ_StepPara:= stStepSend.IQ);
END_METHOD

METHOD PUBLIC m_Senden : BOOL
VAR_INPUT
	I_sTeilenummer		: STRING(19);	// Die Teilenummer die gesendet werden soll
	I_wStatus			: DWORD;			// Der Status des Teils
	I_wZusatzinfo1		: DWORD;			//	Zusätzliche Infos 1
	I_wZusatzinfo2		: DWORD;			// Zusätzliche Infos 2
	I_wZusatzinfo3		: DWORD;			// Zusätzliche Infos 3
	I_wZusatzinfo4		: DWORD;			// Zusätzliche Infos 4
	I_wZusatzinfo5		: DWORD;			//	Zusätzliche Infos 1
	I_wZusatzinfo6		: DWORD;			// Zusätzliche Infos 2
	I_wZusatzinfo7		: DWORD;			// Zusätzliche Infos 3
	I_wZusatzinfo8		: DWORD;			// Zusätzliche Infos 4
	I_wZusatzinfo9		: DWORD;			// Zusätzliche Infos 3
	I_wZusatzinfo10	: DWORD;			// Zusätzliche Infos 4
END_VAR
IF bPartnerLebt
AND Q_bSendeBereit
AND NOT I_bDeaktivieren
THEN
	stTempDatenSend.sTeilenummer		:= I_sTeilenummer;
	stTempDatenSend.wStatus				:= I_wStatus;		
	stTempDatenSend.wZusatzinfo1		:= I_wZusatzinfo1;	
	stTempDatenSend.wZusatzinfo2		:= I_wZusatzinfo2;	
	stTempDatenSend.wZusatzinfo3		:= I_wZusatzinfo3;	
	stTempDatenSend.wZusatzinfo4		:= I_wZusatzinfo4;	
	stTempDatenSend.wZusatzinfo5		:= I_wZusatzinfo5;	
	stTempDatenSend.wZusatzinfo6		:= I_wZusatzinfo6;	
	stTempDatenSend.wZusatzinfo7		:= I_wZusatzinfo7;	
	stTempDatenSend.wZusatzinfo8		:= I_wZusatzinfo8;	
	stTempDatenSend.wZusatzinfo9		:= I_wZusatzinfo9;	
	stTempDatenSend.wZusatzinfo10		:= I_wZusatzinfo10;
	Q_bSendeBereit			:= FALSE;
	stStepSend.IQ.nStep	:= 5;
	m_Senden					:= TRUE;
	
ELSE
	m_Senden					:= FALSE;
END_IF
END_METHOD

END_FUNCTION_BLOCK

// POUs/EAP/FB_EAP_Kommunikation_V2
FUNCTION_BLOCK FB_EAP_Kommunikation_V2
VAR CONSTANT
	nMaxFehlerCounter						: INT := 3;
END_VAR
VAR_INPUT
	I_sNamePartner						: STRING;					// Klartextname der Partneranlage
	I_nFortlaufendeID					: INT;						// Fortlaufende ID
	I_bOhneTwinSAFE					: BOOL;						// Deaktiviert die TwinSAFE Überprüfung und Abarbeitung
	
 	I_nKommBits								: DWORD;					// Kommunikations-Bits aus dem PLC Programm heraus
	I_stTwinSAFEGroupInfoData			: ST_TwinSAFE_Group_Info;	// InfoData der TwinSAFE Gruppe fals TwinSAFE vorhanden
	I_stTwinSAFEConnectionInfoData	: ST_TwinSAFEConnInfo4Byte;// InfoData der TwinSAFE Connection falls vorhanden
	I_bFehlerEtherCAT						: BOOL;						// "glb_bFehler_EtherCATAllg"
	I_bSafetyFreigabe						: BOOL;						// "glb_bSafetyFrg"
		
	{attribute 'hide' := ''}
	I_bDeaktivieren						: BOOL;						// Deaktiviert die Kommunikation sowie die Auswertung
	{attribute 'hide' := ''}
	I_bReset									: BOOL;						// Reset für z.B. anstehende Meldungen
END_VAR
VAR_IN_OUT

	IQ_EAP_Partner_Empfangen			: ST_EAP_Receive;

	IQ_EAP_Partner_Senden				: ST_EAP_Send;
END_VAR
VAR_OUTPUT
	Q_bFehler								: BOOL; 		//Quittierungspflichtiger Fehler liegt an
	Q_bSendeBereit							: BOOL;		// Baustein ist bereit einen neuen Datensatz zu senden
	Q_bNeueDaten							: BOOL;		// Neue Daten von Partner sind vorhanden und können abgerufen werden
	Q_bTwinSAFEReset						: BOOL;		// Quittierungsausgang für zugehörige TwinSAFE Gruppe
	Q_nKommBits								: DWORD;		// Komminkationsbits mit Partneranlage
	Q_bPartnerLebt							: BOOL;		// Verbindung uzm Partner steht
	Q_stDaten								: ST_TempEAPDaten;
	Q_stTwinSAFEConnection				: ST_TwinSAFE_Connection;
	Q_stMeld									: ST_MeldEAPKommError;
													(*	 1 = schlechte Qualität
														 2 = Keine Kommunikation
														 3 = Falsche ID zurückgemeldet oder keine ID
														 4 = TwinSAFE Gruppe in Störung
														 5 = Unbekannter TwinSAFE Fehler
														 6 = TwinSAFE Connection im ungültigen Zustand
														 7 = 
														 8 = 
														 9 = 
														 10 = 
													*)	
	Q_stDatenEmpfangen				: ST_TempEAPDaten;	//Ausgangsstruktur für die empfangenen Daten
	Q_bDatenGesendet					: BOOL;	//Daten wurden Erfolgreich an den Parnter übermittelt
END_VAR
VAR
	bInit									: BOOL;
	arrDatenBuffer						: ARRAY[1..10] OF ST_TempEAPDaten;
	bPartnerLebt						: BOOL;
	
	nStep									: INT;
	nStepSenden							: INT;
	nStepEmpfangen						: INT;
	
	tonTimeOut,
	tonWaitSend,
	tonWaitReceive,
	tonMeldKommError					: TON;
	
	nLastStepSenden					: INT;
	
	nStepBereit,
	nFehlerCounter,
	nIndx									: INT;

	stStepSenden						: ST_StepCtrl;

	bGrpReset							: BOOL;
	tpReset								: TP;
	nLastCycleIndex,
	nLastCycleTOut						: UINT;
	
	stTempDatenSend					: ST_TempEAPDaten;
	
	nOldTwinSAFEGroupMapState,
	nOldTwinSAFEConnectionMapState		: USINT;
	
	sLetzteID							: STRING;	//Letzte erfolgreich gesendete ID
	bFirstCycle							: BOOL;	//Erster Zyklus
	bStartSenden						: BOOL;	//Sendevorgang starten

END_VAR

IF (I_bReset
	AND Q_bFehler)
THEN
	nStep := 0;
END_IF

IF NOT I_bDeaktivieren
THEN
	Q_bPartnerLebt	:=
	bPartnerLebt 	:= 
		NOT tonMeldKommError.Q
		AND (IQ_EAP_Partner_Empfangen.Quality 
			< 4000);
ELSE
	nStep := 0;
END_IF

CASE nStep OF
0: //INIT
	IQ_EAP_Partner_Senden.VarCtrl		 					:= 1;
	IQ_EAP_Partner_Senden.VarData.Data.KommBits		:= 0;
	Q_nKommBits													:= 0;

	stStepSenden.IQ.nStep									:= 0;
	
	IQ_EAP_Partner_Senden.VarData.Data.TeilID			:= '0';
	
	IF NOT I_bDeaktivieren
	THEN
		MEMSET(ADR(stTempDatenSend), 0, SIZEOF(stTempDatenSend));
		MEMSET(ADR(IQ_EAP_Partner_Senden.VarData), 0, SIZEOF(IQ_EAP_Partner_Senden.VarData));
		nStep := 10;
	END_IF
	

10: //Bereit für Kommunikation
	Q_bNeueDaten	:= FALSE;
	IQ_EAP_Partner_Senden.VarCtrl		 				:= 0;
	IQ_EAP_Partner_Senden.VarData.Data.KommBits	:= I_nKommBits;
	
	IF bPartnerLebt
	THEN
		Q_nKommBits		:= IQ_EAP_Partner_Empfangen.VarData.Data.KommBits;
		//_06_Senden();
		//_05_Empfangen();
		_07_Senden_Empfangen();
	ELSE
		Q_bSendeBereit := FALSE;
	END_IF
	
	IF arrDatenBuffer[1].sTeilenummer <> '' 
		AND arrDatenBuffer[1].sTeilenummer <> '0'
		AND arrDatenBuffer[1].wStatus <> 999 //Quittierung Empfang
	THEN
		Q_bNeueDaten	:= TRUE;
	END_IF
	
	IF arrDatenBuffer[1].sTeilenummer <> '' 
		AND arrDatenBuffer[1].sTeilenummer <> '0'
	THEN
		Q_stDatenEmpfangen := arrDatenBuffer[1];

		MEMMOVE(ADR(arrDatenBuffer[1]),ADR(arrDatenBuffer[2]),(SIZEOF(arrDatenBuffer)-SIZEOF(arrDatenBuffer[1])));
		MEMSET(ADR(arrDatenBuffer[10]), 0, SIZEOF(arrDatenBuffer[10]));
	END_IF
	
	IF I_bDeaktivieren
	THEN
		nStep := 0;
	END_IF
	
END_CASE

IF NOT I_bOhneTwinSAFE
THEN
	_02_TwinSAFE();
END_IF

_10_Meldungen();

ACTION _02_TwinSAFE:

IF tonTimeOut.Q
AND NOT I_bFehlerEtherCAT
AND I_bSafetyFreigabe
THEN

	CASE I_stTwinSAFEGroupInfoData.nMapState OF
		1: 
			bGrpReset						:= 
			Q_bTwinSAFEReset				:= 
			Q_stMeld.bMeldTwinSafeGrp		:=
			Q_stMeld.bMeldTwinSafeFehler	:= FALSE;
	
		2..5:
			bGrpReset						:= NOT bGrpReset;
			Q_stMeld.bMeldTwinSafeGrp		:= TRUE;
			
		ELSE
			Q_stMeld.bMeldTwinSafeFehler	:= TRUE;
	END_CASE

(*	// Auswertung Gruppe und Reset
	IF (I_stTwinSAFEGroupInfoData.nMapState
		<> nOldTwinSAFEGroupMapState)
	THEN
		nOldTwinSAFEGroupMapState := I_stTwinSAFEGroupInfoData.nMapState;
		
		CASE I_stTwinSAFEGroupInfoData.nMapState OF
			1: 
				bGrpReset						:= FALSE;
				Q_bTwinSAFEReset				:= FALSE;
				fbMeldung[5].I_bAktiv		:= FALSE;
				fbMeldung[4].I_bAktiv		:= FALSE;	
		
			2..5:
				bGrpReset						:= NOT bGrpReset;
				fbMeldung[4].I_bAktiv		:= TRUE;
				
			ELSE
				fbMeldung[5].I_bAktiv		:= TRUE;
		END_CASE
	END_IF
*)	
	// Auswertung der Connection Info
	IF I_stTwinSAFEConnectionInfoData.nMapState
		<> nOldTwinSAFEConnectionMapState
	THEN
		nOldTwinSAFEConnectionMapState := I_stTwinSAFEConnectionInfoData.nMapState;
		CASE I_stTwinSAFEConnectionInfoData.nMapState OF
			104:	
				Q_stMeld.bMeldTwinSafeUngueltig	:= FALSE;
			ELSE
				Q_stMeld.bMeldTwinSafeUngueltig	:= TRUE;
		END_CASE
	END_IF
END_IF

tpReset(IN := bGrpReset, PT := T#250MS, Q=> Q_bTwinSAFEReset);

Q_stTwinSAFEConnection.Q_bIn0 	:= I_stTwinSAFEConnectionInfoData.nInput.0;
Q_stTwinSAFEConnection.Q_bIn1 	:= I_stTwinSAFEConnectionInfoData.nInput.1;
Q_stTwinSAFEConnection.Q_bIn2 	:= I_stTwinSAFEConnectionInfoData.nInput.2;
Q_stTwinSAFEConnection.Q_bIn3 	:= I_stTwinSAFEConnectionInfoData.nInput.3;
Q_stTwinSAFEConnection.Q_bIn4 	:= I_stTwinSAFEConnectionInfoData.nInput.4;
Q_stTwinSAFEConnection.Q_bIn5 	:= I_stTwinSAFEConnectionInfoData.nInput.5;
Q_stTwinSAFEConnection.Q_bIn6 	:= I_stTwinSAFEConnectionInfoData.nInput.6;
Q_stTwinSAFEConnection.Q_bIn7 	:= I_stTwinSAFEConnectionInfoData.nInput.7;

Q_stTwinSAFEConnection.Q_bOut0 	:= I_stTwinSAFEConnectionInfoData.nOutput.0 AND NOT I_bFehlerEtherCAT;
Q_stTwinSAFEConnection.Q_bOut1 	:= I_stTwinSAFEConnectionInfoData.nOutput.1 AND NOT I_bFehlerEtherCAT;
Q_stTwinSAFEConnection.Q_bOut2 	:= I_stTwinSAFEConnectionInfoData.nOutput.2 AND NOT I_bFehlerEtherCAT;
Q_stTwinSAFEConnection.Q_bOut3 	:= I_stTwinSAFEConnectionInfoData.nOutput.3 AND NOT I_bFehlerEtherCAT;
Q_stTwinSAFEConnection.Q_bOut4 	:= I_stTwinSAFEConnectionInfoData.nOutput.4 AND NOT I_bFehlerEtherCAT;
Q_stTwinSAFEConnection.Q_bOut5 	:= I_stTwinSAFEConnectionInfoData.nOutput.5 AND NOT I_bFehlerEtherCAT;
Q_stTwinSAFEConnection.Q_bOut6 	:= I_stTwinSAFEConnectionInfoData.nOutput.6 AND NOT I_bFehlerEtherCAT;
Q_stTwinSAFEConnection.Q_bOut7 	:= I_stTwinSAFEConnectionInfoData.nOutput.7 AND NOT I_bFehlerEtherCAT;
END_ACTION

ACTION _07_Senden_Empfangen:

//Im ersten Zyklus das Daten gesendet setzen, obwohl noch keine Daten gesendet wurden
IF NOT bFirstCycle
THEN
	Q_bDatenGesendet := TRUE;
	bFirstCycle := TRUE;
END_IF

CASE stStepSenden.IQ.nStep of
	0:	stStepSenden.IQ.sStatus 	:= 'Sendebereit!';
		Q_bSendeBereit 				:= bPartnerLebt;
		Q_stMeld.bMeldFalscheID	:= FALSE;
		
		IQ_EAP_Partner_Senden.VarData.Data.TeilID			:= '0';
		IQ_EAP_Partner_Senden.VarData.Data.TeilStatus	:= 0;
		IQ_EAP_Partner_Senden.VarData.Data.ZusatzInfo1	:= 0;
		IQ_EAP_Partner_Senden.VarData.Data.ZusatzInfo2	:= 0;
		IQ_EAP_Partner_Senden.VarData.Data.ZusatzInfo3	:= 0;
		IQ_EAP_Partner_Senden.VarData.Data.ZusatzInfo4	:= 0;
		IQ_EAP_Partner_Senden.VarData.Data.ZusatzInfo5	:= 0;
		IQ_EAP_Partner_Senden.VarData.Data.ZusatzInfo6	:= 0;
		IQ_EAP_Partner_Senden.VarData.Data.ZusatzInfo7	:= 0;
		IQ_EAP_Partner_Senden.VarData.Data.ZusatzInfo8	:= 0;
		IQ_EAP_Partner_Senden.VarData.Data.ZusatzInfo9	:= 0;
		IQ_EAP_Partner_Senden.VarData.Data.ZusatzInfo10	:= 0;
		
		tonWaitReceive(
			IN := (		 IQ_EAP_Partner_Empfangen.VarData.Data.TeilID <> '0')
						AND(IQ_EAP_Partner_Empfangen.VarData.Data.TeilID <> '')
						AND(IQ_EAP_Partner_Empfangen.VarData.Data.TeilID <>
							 IQ_EAP_Partner_Senden.VarData.Data.TeilID), 
				PT := T#0MS);
		
		//Daten befinden sich im Empfangspuffer
		IF tonWaitReceive.Q
		THEN
			tonWaitReceive(IN:=FALSE);
			stStepSenden.IQ.nStep := 100;
			Q_bSendeBereit							:= FALSE;
			
		//Daten sollen an den Partner gesendet werden
		ELSIF bPartnerLebt
			AND Q_bSendeBereit
			AND stTempDatenSend.sTeilenummer <> ''
			AND stTempDatenSend.sTeilenummer <> '0'
			AND bStartSenden
			//Damit nicht Daten gesendet werden, wenn gerade Daten vom Partner Empfangen wurden
			//Empfangen hat höhere Priorität, für das Quittieren eines Sendevorgangs des dazugehörigen Partners
			AND (IQ_EAP_Partner_Empfangen.VarData.Data.TeilID = '0'
					OR IQ_EAP_Partner_Empfangen.VarData.Data.TeilID = '')
			AND NOT I_bDeaktivieren
		THEN
			stStepSenden.IQ.nStep 		:= 5;
		END_IF
		                           
	5:	stStepSenden.IQ.sStatus 	:= 'Start Senden';
		Q_bSendeBereit 				:= FALSE;
		bStartSenden					:= FALSE;
		
		stStepSenden.IQ.nStep 				:= 10;
		
	10:stStepSenden.IQ.sStatus := 'Kontrolle Sende bereit!';
		tonWaitSend(PT := T#500ms);
		
		IF IQ_EAP_Partner_Senden.FrameState = 0
			AND stTempDatenSend.sTeilenummer <> '0'
			AND stTempDatenSend.sTeilenummer <> ''
			AND stTempDatenSend.sTeilenummer <> IQ_EAP_Partner_Senden.VarData.Data.TeilID
			AND (IQ_EAP_Partner_Empfangen.VarData.Data.TeilID = '0'
					OR IQ_EAP_Partner_Empfangen.VarData.Data.TeilID = '') 
		THEN
			Q_stMeld.bMeldNichtSendebereit	:= FALSE;
			nFehlerCounter					:= 0;
			stStepSenden.IQ.nStep 		:= 15;
		//Damit nicht Daten gesendet werden, wenn gerade Daten vom Partner Empfangen wurden
		//Empfangen hat höhere Priorität, für das Quittieren eines Sendevorgangs
		//Daten wurden in der Empfangsstruktur erkannt und der Sendevorgang wird vorerst abgebrochen damit Daten Empfangen werden können
		ELSIF IQ_EAP_Partner_Empfangen.VarData.Data.TeilID <> '0'
		THEN
			IQ_EAP_Partner_Senden.VarData.Data.TeilID	:= '0';
			stStepSenden.IQ.nStep 		:= 100;
		ELSIF tonWaitSend.Q
		THEN
			nFehlerCounter 			:= nFehlerCounter + 1;
			IF nFehlerCounter > nMaxFehlerCounter
			THEN
				Q_stMeld.bMeldNichtSendebereit	:= TRUE;
				stStepSenden.IQ.nStep 		:= 5;
			END_IF
		END_IF
		
	15:	stStepSenden.IQ.sStatus := 'Daten in Sendebuffer schreiben! RmNr: ';
		stStepSenden.IQ.sStatus := CONCAT( stStepSenden.IQ.sStatus,stTempDatenSend.sTeilenummer);
		stStepSenden.IQ.sStatus := CONCAT( stStepSenden.IQ.sStatus,' Status: ');
		stStepSenden.IQ.sStatus := CONCAT( stStepSenden.IQ.sStatus,DWORD_TO_STRING(stTempDatenSend.wStatus));
 
		//Damit nicht Daten gesendet werden, wenn gerade Daten vom Partner Empfangen wurden
		//Empfangen hat höhere Priorität, für das Quittieren eines Sendevorgangs
		IF (IQ_EAP_Partner_Empfangen.VarData.Data.TeilID = '0'
					OR IQ_EAP_Partner_Empfangen.VarData.Data.TeilID = '') 
		THEN
			IQ_EAP_Partner_Senden.VarData.Data.TeilID				:= stTempDatenSend.sTeilenummer;
			IQ_EAP_Partner_Senden.VarData.Data.TeilStatus		:= stTempDatenSend.wStatus;
			IQ_EAP_Partner_Senden.VarData.Data.ZusatzInfo1		:= stTempDatenSend.wZusatzinfo1;
			IQ_EAP_Partner_Senden.VarData.Data.ZusatzInfo2		:= stTempDatenSend.wZusatzinfo2;
			IQ_EAP_Partner_Senden.VarData.Data.ZusatzInfo3		:= stTempDatenSend.wZusatzinfo3;
			IQ_EAP_Partner_Senden.VarData.Data.ZusatzInfo4		:= stTempDatenSend.wZusatzinfo4;
			IQ_EAP_Partner_Senden.VarData.Data.ZusatzInfo5		:= stTempDatenSend.wZusatzinfo5;
			IQ_EAP_Partner_Senden.VarData.Data.ZusatzInfo6		:= stTempDatenSend.wZusatzinfo6;
			IQ_EAP_Partner_Senden.VarData.Data.ZusatzInfo7		:= stTempDatenSend.wZusatzinfo7;
			IQ_EAP_Partner_Senden.VarData.Data.ZusatzInfo8		:= stTempDatenSend.wZusatzinfo8;
			IQ_EAP_Partner_Senden.VarData.Data.ZusatzInfo9		:= stTempDatenSend.wZusatzinfo9;
			IQ_EAP_Partner_Senden.VarData.Data.ZusatzInfo10		:= stTempDatenSend.wZusatzinfo10;
		//Daten wurden in der Empfangsstruktur erkannt und der Sendevorgang wird vorerst abgebrochen damit Daten Empfangen werden können
		ELSE	
			IQ_EAP_Partner_Senden.VarData.Data.TeilID	:= '0';
			stStepSenden.IQ.nStep 		:= 100;
		END_IF
		
		stStepSenden.IQ.nStep 					:= 20;
		
	20:stStepSenden.IQ.sStatus := 'Kontrolle FrameStaus vorm Senden!';
		tonWaitSend(PT := T#500ms);
		IF IQ_EAP_Partner_Senden.FrameState = 0
			AND (IQ_EAP_Partner_Empfangen.VarData.Data.TeilID = '0'
					OR IQ_EAP_Partner_Empfangen.VarData.Data.TeilID = '')
		THEN
			stStepSenden.IQ.nStep					:= 30;
		//Damit nicht Daten gesendet werden, wenn gerade Daten vom Partner Empfangen wurden
		//Empfangen hat höhere Priorität, für das Quittieren eines Sendevorgangs
		//Daten wurden in der Empfangsstruktur erkannt und der Sendevorgang wird vorerst abgebrochen damit Daten Empfangen werden können
		ELSIF IQ_EAP_Partner_Empfangen.VarData.Data.TeilID <> '0'
		THEN
			IQ_EAP_Partner_Senden.VarData.Data.TeilID	:= '0';
			stStepSenden.IQ.nStep 							:= 100;
		ELSIF tonWaitSend.Q
		THEN
			nFehlerCounter 							:= nFehlerCounter +1;
			Q_stMeld.bMeldNichtSendebereit		:= TRUE;
			stStepSenden.IQ.nStep 					:= 5;
		END_IF
	
	30:	stStepSenden.IQ.sStatus 					:= 'Check Vergleich Senden und Rückmeldung RmNr Senden: ';
		stStepSenden.IQ.sStatus := CONCAT( stStepSenden.IQ.sStatus,IQ_EAP_Partner_Senden.VarData.Data.TeilID) ; 
		stStepSenden.IQ.sStatus := CONCAT( stStepSenden.IQ.sStatus,' RmNr Empfangen: ') ; 
		stStepSenden.IQ.sStatus := CONCAT( stStepSenden.IQ.sStatus,IQ_EAP_Partner_Empfangen.VarData.Data.TeilID) ; 
		tonWaitSend(PT := T#2S);
		
		IF IQ_EAP_Partner_Empfangen.VarData.Data.TeilID =
			IQ_EAP_Partner_Senden.VarData.Data.TeilID
		AND IQ_EAP_Partner_Empfangen.VarData.Data.TeilID <> '0'	
		THEN  
			Q_bDatenGesendet												:= TRUE;	//Daten wurden Erfolgreich übermittelt
			sLetzteID													:= IQ_EAP_Partner_Senden.VarData.Data.TeilID;
			IQ_EAP_Partner_Senden.VarData.Data.TeilID			:= '0';
			IQ_EAP_Partner_Senden.VarData.Data.TeilStatus	:= 0;
			IQ_EAP_Partner_Senden.VarData.Data.ZusatzInfo1	:= 0;
			IQ_EAP_Partner_Senden.VarData.Data.ZusatzInfo2	:= 0;
			IQ_EAP_Partner_Senden.VarData.Data.ZusatzInfo3	:= 0;
			IQ_EAP_Partner_Senden.VarData.Data.ZusatzInfo4	:= 0;
			IQ_EAP_Partner_Senden.VarData.Data.ZusatzInfo5	:= 0;
			IQ_EAP_Partner_Senden.VarData.Data.ZusatzInfo6	:= 0;
			IQ_EAP_Partner_Senden.VarData.Data.ZusatzInfo7	:= 0;
			IQ_EAP_Partner_Senden.VarData.Data.ZusatzInfo8	:= 0;
			IQ_EAP_Partner_Senden.VarData.Data.ZusatzInfo9	:= 0;
			IQ_EAP_Partner_Senden.VarData.Data.ZusatzInfo10	:= 0;
			MEMSET(ADR(stTempDatenSend),0,SIZEOF(stTempDatenSend));
			stStepSenden.IQ.nStep 							:= 40;
			
		//Damit nicht Daten gesendet werden, wenn gerade Daten vom Partner Empfangen wurden
		//Empfangen hat höhere Priorität, für das Quittieren eines Sendevorgangs
		//Daten wurden in der Empfangsstruktur erkannt und der Sendevorgang wird vorerst abgebrochen damit Daten Empfangen werden können
		ELSIF IQ_EAP_Partner_Empfangen.VarData.Data.TeilID <> '0'
			AND IQ_EAP_Partner_Empfangen.VarData.Data.TeilID <> ''
		THEN
			stStepSenden.IQ.nStep 							:= 100;
			
		ELSIF tonWaitSend.Q
		THEN
			Q_stMeld.sErrorID				:= CONCAT('Gesendete ID: ', IQ_EAP_Partner_Senden.VarData.Data.TeilID); 
			stStepSenden.IQ.sStatus 	:= CONCAT( stStepSenden.IQ.sStatus,'Fehler beim Senden Gesendete ID: ') ; 
			stStepSenden.IQ.sStatus 	:= CONCAT( stStepSenden.IQ.sStatus,IQ_EAP_Partner_Senden.VarData.Data.TeilID) ; 
			stStepSenden.IQ.nStep 		:= -30;
		END_IF
		
	40:	stStepSenden.IQ.sStatus 	:= 'Kontrolle FrameStaus nach dem Senden!';
		tonWaitSend(PT := T#500ms);
		IF IQ_EAP_Partner_Senden.FrameState = 0
		THEN
			stStepSenden.IQ.nStep		:= 0;
		END_IF
		
	-30:stStepSenden.IQ.sStatus 					:= 'Fehler beim Senden! Falsche oder keine ID vom Partner zurückgemeldet.';
		Q_stMeld.bMeldFalscheID		:= TRUE;
		IF I_bReset
		THEN
			Q_stMeld.bMeldFalscheID	:= FALSE;
			bStartSenden				:= FALSE;
			stStepSenden.IQ.nStep 	:= 30;
		END_IF
		
	100:stStepSenden.IQ.sStatus := 'Kontrolle Zyklus beim Empfangen!';
		IF IQ_EAP_Partner_Empfangen.CycleIndex <> nLastCycleIndex
		AND bPartnerLebt	
		THEN
			nLastCycleIndex 	:= IQ_EAP_Partner_Empfangen.CycleIndex;
			stStepSenden.IQ.nStep := 110;
		END_IF
		
	110:stStepSenden.IQ.sStatus := 'TeileID: ';
		stStepSenden.IQ.sStatus := CONCAT(stStepSenden.IQ.sStatus, IQ_EAP_Partner_Empfangen.VarData.Data.TeilID);
		stStepSenden.IQ.sStatus := CONCAT(stStepSenden.IQ.sStatus, ' Status: ');
		stStepSenden.IQ.sStatus := CONCAT(stStepSenden.IQ.sStatus, DWORD_TO_STRING(IQ_EAP_Partner_Empfangen.VarData.Data.TeilStatus));
	
		IQ_EAP_Partner_Senden.VarData.Data.TeilID			:= IQ_EAP_Partner_Empfangen.VarData.Data.TeilID;
		IQ_EAP_Partner_Senden.VarData.Data.TeilStatus	:= 999; //Quittierung Empfang
		
		FOR nIndx := 1 TO 10 BY 1 DO
			IF arrDatenBuffer[nIndx].sTeilenummer = ''
				OR arrDatenBuffer[nIndx].sTeilenummer = '0'
			THEN 
				arrDatenBuffer[nIndx].sTeilenummer		:= IQ_EAP_Partner_Empfangen.VarData.Data.TeilID;
				arrDatenBuffer[nIndx].wStatus 			:= IQ_EAP_Partner_Empfangen.VarData.Data.TeilStatus;
				arrDatenBuffer[nIndx].wZusatzinfo1		:= IQ_EAP_Partner_Empfangen.VarData.Data.ZusatzInfo1;
				arrDatenBuffer[nIndx].wZusatzinfo2		:= IQ_EAP_Partner_Empfangen.VarData.Data.ZusatzInfo2;
				arrDatenBuffer[nIndx].wZusatzinfo3		:= IQ_EAP_Partner_Empfangen.VarData.Data.ZusatzInfo3;
				arrDatenBuffer[nIndx].wZusatzinfo4		:= IQ_EAP_Partner_Empfangen.VarData.Data.ZusatzInfo4;
				arrDatenBuffer[nIndx].wZusatzinfo5		:= IQ_EAP_Partner_Empfangen.VarData.Data.ZusatzInfo5;
				arrDatenBuffer[nIndx].wZusatzinfo6		:= IQ_EAP_Partner_Empfangen.VarData.Data.ZusatzInfo6;
				arrDatenBuffer[nIndx].wZusatzinfo7		:= IQ_EAP_Partner_Empfangen.VarData.Data.ZusatzInfo7;
				arrDatenBuffer[nIndx].wZusatzinfo8		:= IQ_EAP_Partner_Empfangen.VarData.Data.ZusatzInfo8;
				arrDatenBuffer[nIndx].wZusatzinfo9		:= IQ_EAP_Partner_Empfangen.VarData.Data.ZusatzInfo9;
				arrDatenBuffer[nIndx].wZusatzinfo10		:= IQ_EAP_Partner_Empfangen.VarData.Data.ZusatzInfo10;
				EXIT;
			END_IF
		END_FOR
		stStepSenden.IQ.nStep								:= 115;
		
	115:stStepSenden.IQ.sStatus := 'Warten aus Teile ID gelöscht!';
		IF IQ_EAP_Partner_Empfangen.VarData.Data.TeilID = '0'
		THEN
			stStepSenden.IQ.nStep							:= 120;
		END_IF
		
	120:stStepSenden.IQ.sStatus := 'Kontrolle Zyklus Empfangen Ende!';
		IF IQ_EAP_Partner_Empfangen.CycleIndex <> nLastCycleIndex
		AND bPartnerLebt
		THEN
			IQ_EAP_Partner_Empfangen.VarData.Data.TeilID := '0';
			IQ_EAP_Partner_Senden.VarData.Data.TeilID	:= '0';
			nLastCycleIndex 									:= IQ_EAP_Partner_Empfangen.CycleIndex;
			stStepSenden.IQ.nStep							:= 0;
		ELSIF NOT Q_bDatenGesendet
			AND bPartnerLebt
			AND IQ_EAP_Partner_Empfangen.CycleIndex <> nLastCycleIndex
		THEN
			nLastCycleIndex 									:= IQ_EAP_Partner_Empfangen.CycleIndex;
			stStepSenden.IQ.nStep							:= 5;
		END_IF
		
END_CASE
stStepSenden.fbHistory(IQ_StepPara:= stStepSenden.IQ);

IF stStepSenden.IQ.nStep <> nLastStepSenden
THEN
	tonWaitSend(IN:=FALSE);
	nLastStepSenden	:= stStepSenden.IQ.nStep;
ELSE
	tonWaitSend(IN:=TRUE);
END_IF
END_ACTION

ACTION _10_Meldungen:
Q_stMeld.sAnlagenteil	:= I_sNamePartner;

tonMeldKommError(IN := (IQ_EAP_Partner_Empfangen.CycleIndex 
									= nLastCycleTOut) ,
						PT := T#500MS);
nLastCycleTOut := IQ_EAP_Partner_Empfangen.CycleIndex;

Q_stMeld.bMeldKommError := 
	tonMeldKommError.Q
	AND NOT I_bDeaktivieren;
		
Q_stMeld.bMeldKeinSignal := 
	IQ_EAP_Partner_Empfangen.Quality 
	> 4000 // Wert erstmal testweise, bei langen Leitungen prüfen ob erhöht werden muss 
	AND NOT Q_stMeld.bMeldKommError
	AND NOT I_bDeaktivieren;
	
	
Q_stMeld.bMeldTwinSafeGrp			:=
Q_stMeld.bMeldTwinSafeFehler		:=
Q_stMeld.bMeldTwinSafeUngueltig	:= FALSE;


Q_bFehler 	:= Q_stMeld.bMeldFalscheID;
END_ACTION

METHOD m_Senden : BOOL
VAR_INPUT
	I_bDeaktivieren	: BOOL;
	
	I_sTeilenummer		: STRING(19);	// Die Teilenummer die gesendet werden soll
	I_wStatus			: DWORD;			// Der Status des Teils
	I_wZusatzinfo1		: DWORD;			//	Zusätzliche Infos 1
	I_wZusatzinfo2		: DWORD;			// Zusätzliche Infos 2
	I_wZusatzinfo3		: DWORD;			// Zusätzliche Infos 3
	I_wZusatzinfo4		: DWORD;			// Zusätzliche Infos 4
	I_wZusatzinfo5		: DWORD;			//	Zusätzliche Infos 1
	I_wZusatzinfo6		: DWORD;			// Zusätzliche Infos 2
	I_wZusatzinfo7		: DWORD;			// Zusätzliche Infos 3
	I_wZusatzinfo8		: DWORD;			// Zusätzliche Infos 4
	I_wZusatzinfo9		: DWORD;			// Zusätzliche Infos 3
	I_wZusatzinfo10	: DWORD;			// Zusätzliche Infos 4
END_VAR

IF bPartnerLebt
	AND Q_bSendeBereit
	AND NOT I_bDeaktivieren
	AND I_sTeilenummer <> '0'
	AND I_sTeilenummer <> ''
THEN
	Q_bSendeBereit := FALSE;
	Q_bDatenGesendet := FALSE;
	bStartSenden	:= TRUE;
	
	stTempDatenSend.sTeilenummer		:= I_sTeilenummer;
	stTempDatenSend.wStatus				:= I_wStatus;		
	stTempDatenSend.wZusatzinfo1		:= I_wZusatzinfo1;	
	stTempDatenSend.wZusatzinfo2		:= I_wZusatzinfo2;	
	stTempDatenSend.wZusatzinfo3		:= I_wZusatzinfo3;	
	stTempDatenSend.wZusatzinfo4		:= I_wZusatzinfo4;	
	stTempDatenSend.wZusatzinfo5		:= I_wZusatzinfo5;	
	stTempDatenSend.wZusatzinfo6		:= I_wZusatzinfo6;	
	stTempDatenSend.wZusatzinfo7		:= I_wZusatzinfo7;	
	stTempDatenSend.wZusatzinfo8		:= I_wZusatzinfo8;	
	stTempDatenSend.wZusatzinfo9		:= I_wZusatzinfo9;	
	stTempDatenSend.wZusatzinfo10		:= I_wZusatzinfo10;
	Q_bSendeBereit							:= FALSE;
END_IF
END_METHOD

END_FUNCTION_BLOCK

// POUs/EAP/FB_StepUebw
{attribute 'reflection'}
FUNCTION_BLOCK FB_StepUebw
VAR_OUTPUT
	//Q_arrStepHist	: ARRAY[1..FB_StepHistory.Q_nMaxStepHistory] OF T_MaxString;
END_VAR
VAR_IN_OUT
	IQ_StepPara		: ST_StepPara;
END_VAR
VAR
	nOldStep			: INT;
	fbStepHistory	: FB_StepHistory;
	tonDelay			: TON;	
	tonAblauf		: TON;	
	
	iZeichen			: INT;
	sBastelPfad		: STRING(255);
	bInit				: BOOL := TRUE;

	{attribute 'instance-path'} 
    {attribute 'noinit'} 
	sPath 			: STRING(255);					// Hier generiert der Compiler beim Systemstart automatisch den Instanzpfad dieser Meldung		
END_VAR


IF bInit THEN
	bInit 		:= FALSE;
	iZeichen 	:= FIND(STR1:= sPath, STR2:= '.');
	sBastelPfad := Delete(STR:= sPath, Len:= iZeichen+1, Pos := 0); 
	iZeichen 	:= FIND(STR1:= sBastelPfad, STR2:= '.');
	sBastelPfad := Delete(STR:= sBastelPfad, Len:= iZeichen+1, Pos := 0);
	
	WHILE FIND(STR1:= sBastelPfad, STR2:= '.')<>0 DO
		sBastelPfad := REPLACE(sBastelPfad,'_',1,FIND(STR1:= sBastelPfad, STR2:= '.'));
	END_WHILE
END_IF
	
	tonDelay(IN:= IQ_StepPara.nStep = nOldStep, PT:= IQ_StepPara.I_tDelay, Q=> IQ_StepPara.Q_bDelay);
	tonAblauf(IN:= IQ_StepPara.I_bAblaufIN, PT:= IQ_StepPara.I_tAblauf, Q=> IQ_StepPara.Q_bAblauf);

	fbStepHistory(
		I_nStep				:= nOldStep );
		
	nOldStep	:= IQ_StepPara.nStep;

END_FUNCTION_BLOCK

// POUs/Logging/FB_StepHistory
FUNCTION_BLOCK FB_StepHistory
VAR CONSTANT
	nMaxStepHistory	:INT	:=	50;
END_VAR
VAR_INPUT
	I_nStep				:INT;
END_VAR
VAR
	n						:INT;
	arrStepHistory		:ARRAY[1..nMaxStepHistory] OF STRING(21);
	nOldHistoryStep	:INT;
END_VAR

	(***********************************************************************)
	IF	I_nStep <> nOldHistoryStep
	THEN
		FOR n := nMaxStepHistory-1  TO 1 BY -1
		DO
			arrStepHistory[n+1] 	:=	arrStepHistory[n];
		END_FOR

		arrStepHistory[1]		:=	INT_TO_STRING(I_nStep);
		FOR n := 5-LEN(arrStepHistory[1]) TO 1 BY -1
		DO
			arrStepHistory[1] := CONCAT(' ', arrStepHistory[1]);
		END_FOR
		arrStepHistory[1] := CONCAT(arrStepHistory[1], ' - ');
		arrStepHistory[1] := CONCAT(arrStepHistory[1], RIGHT(stTimestamp.sQ, 12));

	END_IF

	nOldHistoryStep := I_nStep;

END_FUNCTION_BLOCK

// POUs/EtherCATDiagnose/FB_EtherCATDiag
// FB zur Diagnose des EtherCAT-Masters und aller EtherCAT-Teilnehmer
FUNCTION_BLOCK FB_EtherCATDiag
VAR_IN_OUT
	IQ_stMeldung					: ARRAY [0..cMaxAnzahlSlaveError] OF ST_MeldTextAllgm;
END_VAR
VAR_INPUT
	I_sIPCNetID						: Tc2_System.T_AmsNetID;	// AmsNetId of the IPC x.x.x.x.1.1
	I_sMasterNetID					: Tc2_System.T_AmsNetID;	// AmsNetId of the EtherCAT master device x.x.x.x.2.1
	I_nMasterChangeCnt			: UINT;	// Mit dem EtherCAT Master verknüpfen. ChangeCount
	I_nMasterDevID					: UINT;	// Mit dem EtherCAT Master verknüpfen. Device ID
	I_nSlaveCount 					: UINT;	// Mit dem EtherCAT Master verknüpfen. Anzahl der gefundenen Slaves
	I_nSlaveCountCfg 				: UINT;	// Mit dem EtherCAT Master verknüpfen. Anzahl der konfigurierten und aktivierten Slaves
	I_nMasterDevState				: WORD;	// Mit dem EtherCAT Master verknüpfen. Zustand des EtherCAT-Masters
	I_bAllFrameWcStatesOK		: BOOL;	// Zusammenfassung aller WcStates
	I_tTimeout						: TIME := T#5s;
END_VAR
VAR_OUTPUT
	Q_bEtherCATOK					: BOOL;	// Es liegt ein Fehler im EtherCAT-System vor
	Q_bFrameWcStateError			: BOOL;	// Einer der WcStates ist nicht OK.
	Q_bSlaveCountError			: BOOL;	// Anzahl gefundener Slaves entspricht nicht der Anzahl der knfigurierten ODER keine Slaves gefunden.
	Q_bMasterDevStateError		: BOOL;	// EtherCAT-Master hat einen Error
	Q_bEtherCATSlaveError		: BOOL;	// Ein EtherCAT-Slave hat einen Error
	Q_stMasterDevState			: ST_EcMasterDevState;	// Zustand des EtherCAT-Masters
	Q_bBusy							: BOOL;	// Diagnose durch internen "bDiagReq" gestartet ist in Arbeit
	Q_bError							: BOOL;	// FB-Eingänge nicht richtig beschrieben.
	Q_nErrorID						: UDINT;	// 7: "I_sMasterNetID" nicht korrekt
	
	Q_arrDiagSlaveInfo			: ARRAY [0..3] OF ST_SlaveStateInfo;	// für die Anzeige in der Visu
	Q_arrDiagSlaveInfoScanned	: ARRAY [0..3] OF ST_SlaveStateInfoScanned;	// für die Anzeige in der Visu
END_VAR
VAR
	nState						: INT;	// Index-Variable
	nMasterChangeCntPrev		: UINT;	// zur Erkennung einer EtherCAT-Masteränderung
	nMasterDevStatePrev		: WORD;	// zur Erkennung einer EtherCAT-Master-Zustandsänderung
	bSlaveCountErrorPrev		: BOOL;	// Q_bSlaveCountError über einen Zyklus hinaus speichern, damit die Diagnose nach einem Zustandswechsel nochmal ausgeführt wird.
	bAllFrameWcStatesOKPrev	: BOOL;	// I_bAllFrameWcStatesOK über einen Zyklus hinaus speichern, damit die Diagnose nach einem Zustandswechsel nochmal ausgeführt wird.
	bDiagReq						: BOOL := TRUE;	// Busdiagnose soll ausgeführt werden
	tonDiagReq					: Tc2_Standard.TON;	// Verzögert die Ausführung der Busdiagnose damit nicht ständig diagnostiziert wird.
	n								: DINT;	// Index-Variable

	// Get Slave Addresses
	fbGetSlaveAddresses 		: Tc2_EtherCAT.FB_EcGetAllSlaveAddr;	// Alle online erreichbare EtherCAT-Slave-Adressen holen
	arrSlaveAddresses 		: ARRAY[0..cSlaveAddressArraySize] OF UINT;	// EtherCAT-Adressen aller online erreichbaren Slaves
	nNumOfSlavesRead			: UINT;

	// Get Slave States
	fbGetAllSlaveStates		: Tc2_EtherCAT.FB_EcGetAllSlaveStates;	// Alle online erreichbare EtherCAT-Slave-Adressen holen
	arrSlaveStates 			: ARRAY[0..cSlaveAddressArraySize] OF Tc2_EtherCAT.ST_EcSlaveState;	// EtherCAT-States aller online erreichbaren Slaves

	// Get Topology Data
	nTopologyData				: UDINT;	// Länge/Anzahl der konfigurierten Slaves im Systemmanager
	fbGetTopologyData			: Tc2_System.ADSREAD;
	arrTopologyData			: ARRAY[0..cSlaveAddressArraySize] OF ST_TopologyData;	// Topologiedaten aller EtherCAT-Slaves

	// Check Topology
	arrDiagIndex				: ARRAY [0..3] OF UINT;	// Index im arrTopologyData der Slaves, die an den Ports A bis D hängen. A bzw. 0 ist der eigene Slave
	arrDiagPort					: ARRAY [0..3] OF UINT;	// Slave-Adresse, die an den Ports A bis D hängen. A bzw. 0 ist der eigene Slave
	nIdx							: DINT;	// Index-Variable

	// Scan Slaves
	fbEcGetScannedSlaves		: Tc2_EtherCAT.FB_EcGetScannedSlaves;
	arrScannedSlaveInfo		: ARRAY [0..cSlaveAddressArraySize] OF Tc2_EtherCAT.ST_EcSlaveScannedData;	// Slave Daten. VendorID, ProduktCode, RevisionsNummer, SerialNummer
	nScannedSlaves				: UINT;

	// Get Slave Identities
	fbGetSlaveIdentity		: Tc2_EtherCAT.FB_EcGetSlaveIdentity;
	stIdentity 					: Tc2_EtherCAT.ST_EcSlaveIdentity;

	// Get Slave Names
	fbGetSlaveName 			: Tc2_IoFunctions.IOF_GetBoxNameByAddr;
	sName							: STRING;

	arrSlaveInfo 				: ARRAY [0..cSlaveAddressArraySize] OF ST_SlaveStateInfo;	// EtherCAT-Slave-Infos aus dem Systemmanager (also die konfigurierten Slaves. Nicht die tatsächlich erreichbaren).
	arrSlaveInfoScanned		: ARRAY [0..cSlaveAddressArraySize] OF ST_SlaveStateInfoScanned;	// EtherCAT-Slave-Infos von den erreichbaren EtherCAT-Slaves.

	// Fehlermeldungen
	arrFmEcDiagSlaveError 	: ARRAY [0..cMaxAnzahlSlaveError] OF Tc2_System.T_MaxString;
	nIndexErrorMessage		: INT;
	nIndexSlave					: INT;
END_VAR

//*********************************************************************************************************
// Zyklische Diagnose, FrameError ausgeben. Wird noch woanders ausgewertet, aber hier zusammengefasst.
Q_bFrameWcStateError := NOT I_bAllFrameWcStatesOK;

// Konfigurierte Anzahl an Slaves und gefundene Slaves sind unterschiedlich
Q_bSlaveCountError :=
	(I_nSlaveCount <> I_nSlaveCountCfg)
	OR(I_nSlaveCount= 0);

//*********************************************************************************************************
// Nicht zyklische Diagnose anstoßen, wenn verschiedene Bedingungen erfüllt sind.
//*********************************************************************************************************

// Diagnose anstoßen wenn ein Slave-Anzahl-Fehler aufgefallen ist
IF(Q_bSlaveCountError
		AND NOT bSlaveCountErrorPrev)
	OR(NOT Q_bSlaveCountError
		AND bSlaveCountErrorPrev)
THEN
	bSlaveCountErrorPrev := Q_bSlaveCountError;
	bDiagReq := TRUE;
END_IF

// Diagnose anstoßen wenn nicht alle Framestates OK waren
IF(I_bAllFrameWcStatesOK
		AND NOT bAllFrameWcStatesOKPrev)
	OR(NOT I_bAllFrameWcStatesOK
		AND bAllFrameWcStatesOKPrev)
THEN
	bAllFrameWcStatesOKPrev := I_bAllFrameWcStatesOK;
	bDiagReq := TRUE;
END_IF

// Diagnose anstoßen wenn sich der Zustand des Masters ändert.
// Q_stMasterDevState Updaten
IF(I_nMasterDevState
 <> nMasterDevStatePrev)
THEN
	j_CheckMasterDevState();
	bDiagReq := TRUE;
END_IF

// Diagnose anstoßen wenn sich etwas am Master ändert
IF(I_nMasterChangeCnt
	<> nMasterChangeCntPrev)
THEN
	nMasterChangeCntPrev := I_nMasterChangeCnt;
	bDiagReq := TRUE;
END_IF

//*********************************************************************************************************
// azylische-Diagnose, wird nur bei Änderungen/Fehlern durchgeführt
//*********************************************************************************************************
tonDiagReq(IN	:= bDiagReq, PT:=T#5S);

//*********************************************************************************************************
// azyklische Diagnose ausführen
CASE nState OF
00:	// IDLE, Warten auf Diag start

	IF tonDiagReq.Q
	THEN
		bDiagReq := FALSE;

		IF I_sMasterNetID <> ''
			AND I_sMasterNetID <> '0.0.0.0.0.0'
		THEN	// Diagnose kann beginnen
			nState := nState + 1;
			Q_bBusy := TRUE;
		ELSE
			Q_bError := TRUE;
			Q_nErrorID := 7;
		END_IF

		Q_bEtherCATOK := FALSE;
		
	ELSE
		IF(Q_bSlaveCountError
				OR Q_bMasterDevStateError
				OR NOT I_bAllFrameWcStatesOK)
			AND NOT arrSlaveInfo[arrDiagIndex[0]].bDiagData
		THEN
			Q_bEtherCATOK := FALSE;
			bDiagReq 	:= TRUE;

		ELSIF(Q_bSlaveCountError
				AND NOT bSlaveCountErrorPrev)
			OR (NOT Q_bSlaveCountError
				AND bSlaveCountErrorPrev)
		THEN
			bSlaveCountErrorPrev := Q_bSlaveCountError;
			Q_bEtherCATOK 			:= FALSE;
			bDiagReq 				:= TRUE;

		ELSIF(I_nMasterDevState <> nMasterDevStatePrev)
		THEN
			Q_bEtherCATOK := FALSE;
			bDiagReq 	:= TRUE;

		ELSIF(I_bAllFrameWcStatesOK
				AND NOT bAllFrameWcStatesOKPrev)
			OR (NOT I_bAllFrameWcStatesOK
				AND bAllFrameWcStatesOKPrev)
		THEN
			bAllFrameWcStatesOKPrev := I_bAllFrameWcStatesOK;
			Q_bEtherCATOK 				:= FALSE;
			bDiagReq 					:= TRUE;

		ELSIF Q_bSlaveCountError
				OR Q_bMasterDevStateError
				OR NOT I_bAllFrameWcStatesOK
				OR arrSlaveInfo[arrDiagIndex[0]].bDiagData
		THEN
			Q_bEtherCATOK := FALSE;
		ELSE
			Q_bEtherCATOK := TRUE;
		END_IF
	END_IF

01:	// get adresses
	a_GetSlaveAdresses();
	// nState wird in der Aktion inkrementiert, wenn die Aktion fertig ist.

02:	// get states
	b_GetSlaveStates();
	// nState wird in der Aktion inkrementiert, wenn die Aktion fertig ist.

03:	// get topology data length
	c_GetTopoDataLen();
	// nState wird in der Aktion inkrementiert, wenn die Aktion fertig ist.

04:	// get topology data
	d_GetTopoData();
	// nState wird in der Aktion inkrementiert, wenn die Aktion fertig ist.

05:	// scan online slaves
	e_ScanSlaves();
	// nState wird in der Aktion inkrementiert, wenn die Aktion fertig ist.

06:	// get online identity
	f_GetSlaveIdentity();
	// nState wird in der Aktion inkrementiert, wenn die Aktion fertig ist.

07:	// get name
	g_GetSlaveName();
	// nState wird in der Aktion inkrementiert, wenn die Aktion fertig ist.

08: // get scanned name
	h_GetScannedSlaveName();
	// nState wird in der Aktion inkrementiert, wenn die Aktion fertig ist.

10:	// DONE
	Q_bBusy 	:= FALSE;
	nState 	:= 0;
END_CASE

i_ErrorMessage();

// Fehlermeldungen
FOR n:= 0 TO cMaxAnzahlSlaveError DO
	IF IQ_stMeldung[n].sText <> '' THEN
		IQ_stMeldung[n].bKritFehlerAusg	:= TRUE;
	ELSE
		IQ_stMeldung[n].bKritFehlerAusg	:= FALSE;
	END_IF
END_FOR

// ENDE

ACTION a_GetSlaveAdresses:
//*********************************************************************************************************
// Alle Slave-Adressen der online erreichbaren EtherCAT-Teilnehmer holen

fbGetSlaveAddresses(
	sNetId		:= I_sMasterNetID,
	pAddrBuf		:= ADR(arrSlaveAddresses),
	cbBufLen		:= SIZEOF(arrSlaveAddresses),
	bExecute		:= TRUE,
	tTimeout		:= I_tTimeout,
	nSlaves		=> nNumOfSlavesRead);

IF NOT fbGetSlaveAddresses.bBusy
THEN
	fbGetSlaveAddresses(bExecute:= FALSE);
	
	IF NOT fbGetSlaveAddresses.bError
	THEN
		FOR n := 0 TO MIN(nNumOfSlavesRead, cSlaveAddressArraySize) DO
			arrSlaveInfo[n].nECAddr := arrSlaveAddresses[n];
		END_FOR
	END_IF
	
	nState := nState + 1;	// nächsten Step der Diagnose
	
END_IF

// ENDE
END_ACTION

ACTION b_GetSlaveStates:
//*********************************************************************************************************
// Alle Zustände der online erreichbaren EtherCAT-Teilnehmer holen
fbGetAllSlaveStates(
	sNetId		:= I_sMasterNetID,
	pStateBuf	:= ADR(arrSlaveStates),
	cbBufLen		:= SIZEOF(arrSlaveStates),
	bExecute		:= TRUE,
	tTimeout		:= I_tTimeout,
	nSlaves		=> nNumOfSlavesRead
);

IF NOT fbGetAllSlaveStates.bBusy
THEN
	fbGetAllSlaveStates(bExecute:= FALSE);

	IF NOT fbGetAllSlaveStates.bError
	THEN
		IF nNumOfSlavesRead = I_nSlaveCountCfg
		THEN
			// arrDiagIndex auf 0 setzen
			FOR n := 0 TO 3 DO
				arrDiagIndex[n] := 0;
			END_FOR

			// Die gescannten EtherCAT-Slave-States in die Info-Struktur "arrSlaveInfo" schreiben
			FOR n := 0 TO MIN(nNumOfSlavesRead, cSlaveAddressArraySize) DO
				// EtherCAT-Slave-State
				arrSlaveInfo[n].stState.eEcState 			:= arrSlaveStates[n].deviceState AND 16#0F;
				arrSlaveInfo[n].stState.bError 				:= arrSlaveStates[n].deviceState.4;
				arrSlaveInfo[n].stState.bInvalidVPRS 		:= arrSlaveStates[n].deviceState.5;
				// EtherCAT-Link-State
				arrSlaveInfo[n].stState.bNoCommToSlave 	:= arrSlaveStates[n].linkState.0;
				arrSlaveInfo[n].stState.bLinkError 			:= arrSlaveStates[n].linkState.1;
				arrSlaveInfo[n].stState.bMissingLink 		:= arrSlaveStates[n].linkState.2;
				arrSlaveInfo[n].stState.bUnexpectedLink	:= arrSlaveStates[n].linkState.3;
				arrSlaveInfo[n].stState.bPortA 				:= arrSlaveStates[n].linkState.4;
				arrSlaveInfo[n].stState.bPortB 				:= arrSlaveStates[n].linkState.5;
				arrSlaveInfo[n].stState.bPortC 				:= arrSlaveStates[n].linkState.6;
				arrSlaveInfo[n].stState.bPortD 				:= arrSlaveStates[n].linkState.7;
				// bDiagData zuweisen, wenn Diagnosedaten vorhanden sind.
				arrSlaveInfo[n].bDiagData	:=
					((arrSlaveStates[n].deviceState AND 16#F0) <> 0)
						OR (((arrSlaveStates[n].deviceState AND 16#0F) > 0)
							AND ((arrSlaveStates[n].deviceState AND 16#0F) < 8))
					OR (arrSlaveStates[n].linkState <> 0);

				IF arrSlaveInfo[n].bDiagData
				THEN	// Aktueller Slave hat Diagnosedaten, es gibt also einen Fehler!
					IF (n=0)
					THEN	// n=0 ist der Master. Der wird einfach auf 0 gesetzt
						arrDiagIndex[0] := 0;
					ELSE
						IF (arrDiagIndex[0] = 0)
							AND NOT arrSlaveInfo[0].bDiagData
						THEN
							arrDiagIndex[0] :=  DINT_TO_UINT(n);	// Arrayindex vom 1. arrSlaveInfo speichern, an dem Diagnose-Daten vorhanden sind.
						END_IF
					END_IF
				END_IF
				
			END_FOR
		END_IF
	END_IF

	IF arrSlaveInfo[arrDiagIndex[0]].bDiagData
	THEN	// Wenn ein Diagnosedatum gefunden wurde, wird der state weitergeschaltet
		nState := nState + 1;
	ELSE	// Wenn keine Diagnosedaten gefunden wurden, wedern die Ausgänge auf 0 gesetzt und im Schritt nach 10. Damit wäre die Diagnose durch
		FOR n := 0 TO 3 DO
			MEMSET(ADR(Q_arrDiagSlaveInfo[n]), 0, SIZEOF(Q_arrDiagSlaveInfo[n]));
			MEMSET(ADR(Q_arrDiagSlaveInfoScanned[n]), 0, SIZEOF(Q_arrDiagSlaveInfoScanned[n]));
		END_FOR
		nState := 10;
	END_IF
END_IF

// ENDE
END_ACTION

ACTION c_GetTopoDataLen:
//*********************************************************************************************************
// Anzahl der Teilnehmer in der EtherCAT-Topologie der aktiven Konfiguration auslesen
fbGetTopologyData(
	NETID			:= I_sMasterNetID,
	PORT			:= 16#FFFF,
	IDXGRP		:= EC_ADS_IGRP_MASTER_COUNT_SLAVE,
	IDXOFFS		:= EC_ADS_IOFFS_MASTER_COUNT_SLAVE,
	LEN			:= SIZEOF(nTopologyData),
	DESTADDR		:= ADR(nTopologyData),
	READ			:= TRUE,
	TMOUT			:= I_tTimeout
);

IF NOT fbGetTopologyData.BUSY
THEN
	fbGetTopologyData(READ := FALSE);
	nState := nState + 1;
END_IF

// ENDE
END_ACTION

ACTION d_GetTopoData:
//*********************************************************************************************************
// EtherCAT-Topologiedaten aus der aktivierten Konfiguration holen
fbGetTopologyData(
	NETID			:= I_sMasterNetID,
	PORT			:= 16#FFFF,
	IDXGRP		:= 16#22,
	IDXOFFS		:= 0,
	LEN			:= nTopologyData*SIZEOF(arrTopologyData[0]),
	DESTADDR		:= ADR(arrTopologyData),
	READ			:= TRUE,
	TMOUT			:= I_tTimeout
);

IF NOT fbGetTopologyData.BUSY
THEN
	fbGetTopologyData(READ := FALSE);

	IF NOT fbGetTopologyData.ERR
	THEN
		// In arrDiagIndex[0] ist der erste Index aller EtherCAT-Slaves mit einer Diagnosemeldung enthalten
		// Adressen an dem ersten EtherCAT-Slave mit Diagnosemeldung speichern
		arrDiagPort[0] := arrTopologyData[arrDiagIndex[0]].nOwnPhysicalAddr;
		arrDiagPort[1] := arrTopologyData[arrDiagIndex[0]].stPhysicalAddr.nPortB;
		arrDiagPort[2] := arrTopologyData[arrDiagIndex[0]].stPhysicalAddr.nPortC;
		arrDiagPort[3] := arrTopologyData[arrDiagIndex[0]].stPhysicalAddr.nPortD;

		// erstmal alle weiteren Indexe auf 0 setzen
		arrDiagIndex[1] := 0;
		arrDiagIndex[2] := 0;
		arrDiagIndex[3] := 0;

		// Index des EtherCAT-Slaves am Port B suchen
		IF arrDiagPort[1] <> 0
		THEN
			FOR n := 0 TO MIN(UDINT_TO_DINT(nTopologyData)-1,cSlaveAddressArraySize) DO
				IF arrTopologyData[n].nOwnPhysicalAddr = arrDiagPort[1]
				THEN
					arrDiagIndex[1] :=  DINT_TO_UINT(n);
					EXIT;
				END_IF
			END_FOR
		END_IF

		// Index des EtherCAT-Slaves am Port C suchen
		IF arrDiagPort[2] <> 0
		THEN
			FOR n := 0 TO MIN(UDINT_TO_DINT(nTopologyData)-1,cSlaveAddressArraySize) DO
				IF arrTopologyData[n].nOwnPhysicalAddr = arrDiagPort[2]
				THEN
					arrDiagIndex[2] :=  DINT_TO_UINT(n);
					EXIT;
				END_IF
			END_FOR
		END_IF

		// Index des EtherCAT-Slaves am Port D suchen
		IF arrDiagPort[3] <> 0
		THEN
			FOR n := 0 TO MIN(UDINT_TO_DINT(nTopologyData)-1,cSlaveAddressArraySize) DO
				IF arrTopologyData[n].nOwnPhysicalAddr = arrDiagPort[3]
				THEN
					arrDiagIndex[3] :=  DINT_TO_UINT(n);
					EXIT;
				END_IF
			END_FOR
		END_IF
		
	END_IF

	nIdx := 0;
	nState := nState + 1;
	
END_IF

// ENDE
END_ACTION

ACTION e_ScanSlaves:
//*********************************************************************************************************
// Infodaten von Online erreichbaren Slaves holen.
fbEcGetScannedSlaves(
	bExecute						:= TRUE,
	sNetId						:= I_sMasterNetID,
	pArrEcScannedSlaveInfo	:= ADR(arrScannedSlaveInfo),
	cbBufLen						:= SIZEOF(arrScannedSlaveInfo),
	tTimeout						:= I_tTimeout
);

IF NOT fbEcGetScannedSlaves.bBusy
THEN
	fbEcGetScannedSlaves(bExecute := FALSE);
	nState := nState + 1;

	IF fbEcGetScannedSlaves.bError
	THEN
		nScannedSlaves := 0;
	ELSE
		nScannedSlaves := fbEcGetScannedSlaves.nSlaves;
	END_IF
	
END_IF

// ENDE
END_ACTION

ACTION f_GetSlaveIdentity:
//*********************************************************************************************************
// Systemmanager-Typ des Slaves mit der Diagnosemeldung holen. Z.B.: EL1002
fbGetSlaveIdentity(
	sNetId		:= I_sMasterNetID,
	nSlaveAddr	:= arrSlaveInfo[arrDiagIndex[nIdx]].nECAddr,
	bExecute		:= TRUE,
	tTimeout		:= I_tTimeout,
	identity		=> stIdentity
);

IF NOT fbGetSlaveIdentity.bBusy
THEN
	fbGetSlaveIdentity(bExecute:= FALSE);

	IF NOT fbGetSlaveIdentity.bError
	THEN
		IF arrDiagPort[nIdx] <> 0
		THEN
			arrSlaveInfo[arrDiagIndex[nIdx]].nIndex	:= arrDiagIndex[nIdx] + 1;
			arrSlaveInfo[arrDiagIndex[nIdx]].sType 	:= F_ConvProductCodeToString(stSlaveIdentity := stIdentity);
		END_IF
	END_IF
	
	nState := nState + 1;
	
END_IF

// ENDE
END_ACTION

ACTION g_GetSlaveName:
//*********************************************************************************************************
// Systemmanager-Namen des Slaves mit der Diagnosemeldung holen. Z.B.: "=S20.7-BC1"
fbGetSlaveName(
	NETID			:= I_sIPCNetID,
	DEVICEID		:= I_nMasterDevID,
	BOXADDR		:= arrSlaveInfo[arrDiagIndex[nIdx]].nECAddr,
	START			:= TRUE,
	TMOUT			:= I_tTimeout,
	BOXNAME		=> sName
);

IF NOT fbGetSlaveName.BUSY
THEN
	fbGetSlaveName(START:= FALSE);

	IF NOT fbGetSlaveName.ERR
	THEN
		IF arrDiagPort[nIdx] <> 0
		THEN
			arrSlaveInfo[arrDiagIndex[nIdx]].sName 	:= sName;
		END_IF
	END_IF

	nState := nState + 1;
	
END_IF

// ENDE
END_ACTION

ACTION h_GetScannedSlaveName:
//*********************************************************************************************************
// Slave-Namen des Online erreichbaren Slaves mit einer Diagnosemeldung ist abgleichen
// arrDiagIndex[nIdx] sind Slaves mit Diagnosemeldung
fbGetSlaveName(
	NETID			:= I_sIPCNetID,
	DEVICEID		:= I_nMasterDevID,
	BOXADDR		:= arrScannedSlaveInfo[arrDiagIndex[nIdx]].nAddr,
	START			:= TRUE,
	TMOUT			:= I_tTimeout,
	BOXNAME		=> sName
);

IF NOT fbGetSlaveName.BUSY
THEN
	fbGetSlaveName(START:= FALSE);

	(* add scanned info *)
	arrSlaveInfoScanned[arrDiagIndex[nIdx]].nIndex 	:= arrDiagIndex[nIdx] + 1;

	IF arrScannedSlaveInfo[arrDiagIndex[nIdx]].nAddr <> 0
	THEN
		IF NOT fbGetSlaveName.ERR
		THEN
			arrSlaveInfoScanned[arrDiagIndex[nIdx]].sName := sName;
		END_IF
	ELSE
		arrSlaveInfoScanned[arrDiagIndex[nIdx]].sType		:= '';
	END_IF

	IF (arrDiagIndex[nIdx] < nScannedSlaves)
	THEN
		arrSlaveInfoScanned[arrDiagIndex[nIdx]].sType		:= F_ConvProductCodeToString(arrScannedSlaveInfo[arrDiagIndex[nIdx]].stSlaveIdentity);
	ELSE
		arrSlaveInfoScanned[arrDiagIndex[nIdx]].sType		:= '';
	END_IF

	arrSlaveInfoScanned[arrDiagIndex[nIdx]].nECAddr		:= arrScannedSlaveInfo[arrDiagIndex[nIdx]].nAddr;

	IF arrSlaveInfoScanned[arrDiagIndex[nIdx]].sName <> arrSlaveInfo[arrDiagIndex[nIdx]].sName
	THEN
		arrSlaveInfoScanned[arrDiagIndex[nIdx]].bDifferentName := TRUE;
	ELSE
		arrSlaveInfoScanned[arrDiagIndex[nIdx]].bDifferentName := FALSE;
	END_IF

	IF arrSlaveInfoScanned[arrDiagIndex[nIdx]].nECAddr <> arrSlaveInfo[arrDiagIndex[nIdx]].nECAddr
	THEN
		arrSlaveInfoScanned[arrDiagIndex[nIdx]].bDifferentAddr := TRUE;
	ELSE
		arrSlaveInfoScanned[arrDiagIndex[nIdx]].bDifferentAddr := FALSE;
	END_IF

	IF arrSlaveInfoScanned[arrDiagIndex[nIdx]].sType <> arrSlaveInfo[arrDiagIndex[nIdx]].sType
	THEN
		arrSlaveInfoScanned[arrDiagIndex[nIdx]].bDifferentType := TRUE;
	ELSE
		arrSlaveInfoScanned[arrDiagIndex[nIdx]].bDifferentType := FALSE;
	END_IF

	IF nIdx < 3
	THEN
		nIdx := nIdx + 1;
		nState := nState - 2;
	ELSE	// wenn nIdx = 3 ist, werden die letzten 3 Aktionen nicht wiederholt und die Fehler an die Ausgänge übergeben
		nIdx := 0;
		nState := 10;

		FOR n := 0 TO 3 DO
			IF arrDiagPort[n] <> 0
			THEN	// Meldungen füllen
				Q_arrDiagSlaveInfo[n] := arrSlaveInfo[arrDiagIndex[n]];
				Q_arrDiagSlaveInfoScanned[n] := arrSlaveInfoScanned[arrDiagIndex[n]];
			ELSE
				MEMSET(ADR(Q_arrDiagSlaveInfo[n]), 0, SIZEOF(Q_arrDiagSlaveInfo[n]));
				MEMSET(ADR(Q_arrDiagSlaveInfoScanned[n]), 0, SIZEOF(Q_arrDiagSlaveInfoScanned[n]));
			END_IF
		END_FOR
	END_IF
END_IF

(*BE*)
END_ACTION

ACTION i_ErrorMessage:
//*********************************************************************************************************
// Fehlermeldungen zusammenfassen und in STRINGs packen
//*********************************************************************************************************

// Fehlermeldungen löschen
FOR nIndexErrorMessage := 0  TO cMaxAnzahlSlaveError DO
	IQ_stMeldung[nIndexErrorMessage].sText	:= '';
END_FOR

nIndexErrorMessage := 0;

//*********************************************************************************************************
// Fehler bei Anzahl der Teilnehmer
IF Q_bSlaveCountError
THEN

	IQ_stMeldung[nIndexErrorMessage].SourceName	:= 'EtherCAT-Bus';

	IQ_stMeldung[nIndexErrorMessage].sText :=
		CONCAT(	'Anzahl der konfigurierten Teilnehmer: ',
					UINT_TO_STRING(I_nSlaveCountCfg));

	IQ_stMeldung[nIndexErrorMessage].sText :=
		CONCAT(	IQ_stMeldung[nIndexErrorMessage].sText,
					' , Anzahl der erkannten Teilnehmer: ');

	IQ_stMeldung[nIndexErrorMessage].sText :=
		CONCAT(	IQ_stMeldung[nIndexErrorMessage].sText,
					UINT_TO_STRING(I_nSlaveCount));

	IQ_stMeldung[nIndexErrorMessage].sText :=
		CONCAT(	IQ_stMeldung[nIndexErrorMessage].sText,
					' !');

	IF nIndexErrorMessage < cMaxAnzahlSlaveError
	THEN
		nIndexErrorMessage := nIndexErrorMessage + 1;
	ELSE
		RETURN;
	END_IF
END_IF

//*********************************************************************************************************
// Status-Informationen - DevState RT Ethernet Adapter
IF Q_stMasterDevState.bLinkError THEN
	
	IQ_stMeldung[nIndexErrorMessage].SourceName	:=	'EtherCAT-Bus';
	IQ_stMeldung[nIndexErrorMessage].sText := 'Status: Link Error (Netzwerkverbindung physikalisch unterbrochen) !';

	IF nIndexErrorMessage < cMaxAnzahlSlaveError THEN
		nIndexErrorMessage := nIndexErrorMessage + 1;
	ELSE
		RETURN;
	END_IF
END_IF

(* --- *)
IF Q_stMasterDevState.bResetActive THEN
	
	IQ_stMeldung[nIndexErrorMessage].SourceName	:=	'EtherCAT-Bus';
	IQ_stMeldung[nIndexErrorMessage].sText := 'Status: I/O-Reset ist aktiv !';
	IF nIndexErrorMessage < cMaxAnzahlSlaveError THEN
		nIndexErrorMessage := nIndexErrorMessage + 1;
	ELSE
		RETURN;
	END_IF
END_IF

(* --- *)
IF Q_stMasterDevState.bAtLeastOneNotInOp THEN

	IQ_stMeldung[nIndexErrorMessage].SourceName	:=	'EtherCAT-Bus';
	IQ_stMeldung[nIndexErrorMessage].sText := 'Status: Mindestens ein Teilnehmer ist nicht im OP-State (Betriebsbereit) !';

	IF nIndexErrorMessage < cMaxAnzahlSlaveError THEN
		nIndexErrorMessage := nIndexErrorMessage + 1;
	ELSE
		RETURN;
	END_IF
END_IF

(* --- *)

IF Q_stMasterDevState.bDcNotInSync THEN
	
	IQ_stMeldung[nIndexErrorMessage].SourceName	:=	'EtherCAT-Bus';
	IQ_stMeldung[nIndexErrorMessage].sText := 'Status: Distributed Clocks sind nicht synchronisiert / im Zeitfenster !';

	IF nIndexErrorMessage < cMaxAnzahlSlaveError THEN
		nIndexErrorMessage := nIndexErrorMessage + 1;
	ELSE
		RETURN;
	END_IF
END_IF

(* --- *)

IF Q_stMasterDevState.bDriverNotFound THEN
	
	IQ_stMeldung[nIndexErrorMessage].SourceName	:=	'EtherCAT-Bus';
	IQ_stMeldung[nIndexErrorMessage].sText := 'Status: TwinCAT Real-Time Ethernet Treiber nicht gefunden !';

	IF nIndexErrorMessage < cMaxAnzahlSlaveError THEN
		nIndexErrorMessage := nIndexErrorMessage + 1;
	ELSE
		RETURN;
	END_IF
END_IF

(* --- *)

IF (I_nMasterDevState AND 16#000F) = 2 THEN
	
	IQ_stMeldung[nIndexErrorMessage].SourceName	:=	'EtherCAT-Bus';
	IQ_stMeldung[nIndexErrorMessage].sText := 'Status: E/A gesperrt nach Link Error (E/A Reset notwendig nach Behebung) !';

	IF nIndexErrorMessage < cMaxAnzahlSlaveError THEN
		nIndexErrorMessage := nIndexErrorMessage + 1;
	ELSE
		RETURN;
	END_IF
END_IF

(* --- *)

IF (I_nMasterDevState AND 16#FFF0) = 16#10 THEN
	
	IQ_stMeldung[nIndexErrorMessage].SourceName	:=	'EtherCAT-Bus';
	IQ_stMeldung[nIndexErrorMessage].sText := 'Status: Keine Senderesourcen vorhanden (E/A Reset notwendig nach Behebung) !';

	IF nIndexErrorMessage < cMaxAnzahlSlaveError THEN
		nIndexErrorMessage := nIndexErrorMessage + 1;
	ELSE
		RETURN;
	END_IF
END_IF

(* --- *)

IF Q_stMasterDevState.bWatchdogTriggerd THEN
	
	IQ_stMeldung[nIndexErrorMessage].SourceName	:=	'EtherCAT-Bus';
	IQ_stMeldung[nIndexErrorMessage].sText := 'Status: Watchdog hat zugeschlagen !';

	IF nIndexErrorMessage < cMaxAnzahlSlaveError THEN
		nIndexErrorMessage := nIndexErrorMessage + 1;
	ELSE
		RETURN;
	END_IF
END_IF

(* --- *)

IF Q_stMasterDevState.bMissFrmRedMode THEN
	
	IQ_stMeldung[nIndexErrorMessage].SourceName	:=	'EtherCAT-Bus';
	IQ_stMeldung[nIndexErrorMessage].sText := 'Status: Missing one frame !';

	IF nIndexErrorMessage < cMaxAnzahlSlaveError THEN
		nIndexErrorMessage := nIndexErrorMessage + 1;
	ELSE
		RETURN;
	END_IF
END_IF

//*********************************************************************************************************
IF Q_arrDiagSlaveInfo[0].bDiagData
THEN

	(* CRC-Fehler ------------------------------------------------------------------------- *)
	(* Anzahl der CRC-Fehler am Port A *)
	IF Q_arrDiagSlaveInfo[0].stPortCRCErrors.portA > 0 THEN

			IQ_stMeldung[nIndexErrorMessage].SourceName	:=	'EtherCAT-Bus';
			IQ_stMeldung[nIndexErrorMessage].sText :=
				CONCAT(	'Status EtherCAT-Bus: Teilnehmer: ',
							Q_arrDiagSlaveInfo[0].sName);

			IQ_stMeldung[nIndexErrorMessage].sText :=
				CONCAT(	IQ_stMeldung[nIndexErrorMessage].sText,
							', Typ: ');

			IQ_stMeldung[nIndexErrorMessage].sText :=
				CONCAT(	IQ_stMeldung[nIndexErrorMessage].sText,
							Q_arrDiagSlaveInfo[0].sType);

			IQ_stMeldung[nIndexErrorMessage].sText :=
				CONCAT(	IQ_stMeldung[nIndexErrorMessage].sText,
							': Anzahl der CRC-Fehler am Port A: ');

			IQ_stMeldung[nIndexErrorMessage].sText :=
				CONCAT(	IQ_stMeldung[nIndexErrorMessage].sText,
							UDINT_TO_STRING(Q_arrDiagSlaveInfo[0].stPortCRCErrors.portA));
	END_IF

	(* Anzahl der CRC-Fehler am Port B *)
	IF Q_arrDiagSlaveInfo[0].stPortCRCErrors.portB > 0 THEN

			IQ_stMeldung[nIndexErrorMessage].SourceName	:=	'EtherCAT-Bus';
			IQ_stMeldung[nIndexErrorMessage].sText :=
				CONCAT(	'Status EtherCAT-Bus: Teilnehmer: ',
							Q_arrDiagSlaveInfo[0].sName);

			IQ_stMeldung[nIndexErrorMessage].sText :=
				CONCAT(	IQ_stMeldung[nIndexErrorMessage].sText,
							', Typ: ');

			IQ_stMeldung[nIndexErrorMessage].sText :=
				CONCAT(	IQ_stMeldung[nIndexErrorMessage].sText,
							Q_arrDiagSlaveInfo[0].sType);

			IQ_stMeldung[nIndexErrorMessage].sText :=
				CONCAT(	IQ_stMeldung[nIndexErrorMessage].sText,
							': Anzahl der CRC-Fehler am Port B: ');

			IQ_stMeldung[nIndexErrorMessage].sText :=
				CONCAT(	IQ_stMeldung[nIndexErrorMessage].sText,
							UDINT_TO_STRING(Q_arrDiagSlaveInfo[0].stPortCRCErrors.portB));
	END_IF

	(* Anzahl der CRC-Fehler am Port C *)
	IF Q_arrDiagSlaveInfo[0].stPortCRCErrors.portC > 0 THEN

			IQ_stMeldung[nIndexErrorMessage].SourceName	:=	'EtherCAT-Bus';
			IQ_stMeldung[nIndexErrorMessage].sText :=
				CONCAT(	'Status EtherCAT-Bus: Teilnehmer: ',
							Q_arrDiagSlaveInfo[0].sName);

			IQ_stMeldung[nIndexErrorMessage].sText :=
				CONCAT(	IQ_stMeldung[nIndexErrorMessage].sText,
							', Typ: ');

			IQ_stMeldung[nIndexErrorMessage].sText :=
				CONCAT(	IQ_stMeldung[nIndexErrorMessage].sText,
							Q_arrDiagSlaveInfo[0].sType);

			IQ_stMeldung[nIndexErrorMessage].sText :=
				CONCAT(	IQ_stMeldung[nIndexErrorMessage].sText,
							': Anzahl der CRC-Fehler am Port C: ');

			IQ_stMeldung[nIndexErrorMessage].sText :=
				CONCAT(	IQ_stMeldung[nIndexErrorMessage].sText,
							UDINT_TO_STRING(Q_arrDiagSlaveInfo[0].stPortCRCErrors.portC));
	END_IF

	(* Anzahl der CRC-Fehler am Port D *)
	IF Q_arrDiagSlaveInfo[0].stPortCRCErrors.portD > 0 THEN

			IQ_stMeldung[nIndexErrorMessage].SourceName	:=	'EtherCAT-Bus';
			IQ_stMeldung[nIndexErrorMessage].sText :=
				CONCAT(	'Status EtherCAT-Bus: Teilnehmer: ',
							Q_arrDiagSlaveInfo[0].sName);

			IQ_stMeldung[nIndexErrorMessage].sText :=
				CONCAT(	IQ_stMeldung[nIndexErrorMessage].sText,
							', Typ: ');

			IQ_stMeldung[nIndexErrorMessage].sText :=
				CONCAT(	IQ_stMeldung[nIndexErrorMessage].sText,
							Q_arrDiagSlaveInfo[0].sType);

			IQ_stMeldung[nIndexErrorMessage].sText :=
				CONCAT(	IQ_stMeldung[nIndexErrorMessage].sText,
							': Anzahl der CRC-Fehler am Port D: ');

			IQ_stMeldung[nIndexErrorMessage].sText :=
				CONCAT(	IQ_stMeldung[nIndexErrorMessage].sText,
							UDINT_TO_STRING(Q_arrDiagSlaveInfo[0].stPortCRCErrors.portD));
	END_IF

	(* ------------------------------------------------------------------------------------ *)

	CASE Q_arrDiagSlaveInfo[0].stState.eEcState OF

	eEcState_OP:
		(* Link am angegebenen Port fehlt (Port = A, B, C or D) *)
		IF Q_arrDiagSlaveInfo[0].stState.bMissingLink THEN

			IQ_stMeldung[nIndexErrorMessage].SourceName	:=	'EtherCAT-Bus';
			IQ_stMeldung[nIndexErrorMessage].sText :=
				CONCAT(	'Fehler EtherCAT-Bus: Teilnehmer: ',
							Q_arrDiagSlaveInfo[0].sName);

			IQ_stMeldung[nIndexErrorMessage].sText :=
				CONCAT(	IQ_stMeldung[nIndexErrorMessage].sText,
							', Typ: ');

			IQ_stMeldung[nIndexErrorMessage].sText :=
				CONCAT(	IQ_stMeldung[nIndexErrorMessage].sText,
							Q_arrDiagSlaveInfo[0].sType);

			IF Q_arrDiagSlaveInfo[0].stState.bPortA THEN
					IQ_stMeldung[nIndexErrorMessage].sText :=
						CONCAT(	IQ_stMeldung[nIndexErrorMessage].sText,
									': Link am Port A fehlt !');
			ELSIF Q_arrDiagSlaveInfo[0].stState.bPortB THEN
				IQ_stMeldung[nIndexErrorMessage].sText :=
					CONCAT(	IQ_stMeldung[nIndexErrorMessage].sText,
								': Link am Port B fehlt !');
			ELSIF Q_arrDiagSlaveInfo[0].stState.bPortC THEN
				IQ_stMeldung[nIndexErrorMessage].sText :=
					CONCAT(	IQ_stMeldung[nIndexErrorMessage].sText,
								': Link am Port C fehlt !');
			ELSIF Q_arrDiagSlaveInfo[0].stState.bPortD THEN
				IQ_stMeldung[nIndexErrorMessage].sText :=
					CONCAT(	IQ_stMeldung[nIndexErrorMessage].sText,
								': Link am Port D fehlt !');
			END_IF

			IF nIndexErrorMessage < cMaxAnzahlSlaveError THEN
				nIndexErrorMessage := nIndexErrorMessage + 1;
			ELSE
				RETURN;
			END_IF

		(* Ein zusätzlicher Link wurde am angegebenen Port festgestellt *)
		ELSIF Q_arrDiagSlaveInfo[0].stState.bUnexpectedLink THEN

			IQ_stMeldung[nIndexErrorMessage].SourceName	:=	'EtherCAT-Bus';
			IQ_stMeldung[nIndexErrorMessage].sText :=
				CONCAT(	'Fehler EtherCAT-Bus: Teilnehmer: ',
							Q_arrDiagSlaveInfo[0].sName);

			IQ_stMeldung[nIndexErrorMessage].sText :=
				CONCAT(	IQ_stMeldung[nIndexErrorMessage].sText,
							', Typ: ');

			IQ_stMeldung[nIndexErrorMessage].sText :=
				CONCAT(	IQ_stMeldung[nIndexErrorMessage].sText,
							Q_arrDiagSlaveInfo[0].sType);

			IF Q_arrDiagSlaveInfo[0].stState.bPortA THEN
				IQ_stMeldung[nIndexErrorMessage].sText :=
						CONCAT(	IQ_stMeldung[nIndexErrorMessage].sText,
									': Ein zusätzlicher Link wurde am Port A festgestellt !');
			ELSIF Q_arrDiagSlaveInfo[0].stState.bPortB THEN
				IQ_stMeldung[nIndexErrorMessage].sText :=
					CONCAT(	IQ_stMeldung[nIndexErrorMessage].sText,
									': Ein zusätzlicher Link wurde am Port B festgestellt !');
			ELSIF Q_arrDiagSlaveInfo[0].stState.bPortC THEN
				IQ_stMeldung[nIndexErrorMessage].sText :=
					CONCAT(	IQ_stMeldung[nIndexErrorMessage].sText,
									': Ein zusätzlicher Link wurde am Port C festgestellt !');
			ELSIF Q_arrDiagSlaveInfo[0].stState.bPortD THEN
				IQ_stMeldung[nIndexErrorMessage].sText :=
					CONCAT(	IQ_stMeldung[nIndexErrorMessage].sText,
									': Ein zusätzlicher Link wurde am Port D festgestellt !');
			END_IF

			IF nIndexErrorMessage < cMaxAnzahlSlaveError THEN
				nIndexErrorMessage := nIndexErrorMessage + 1;
			ELSE
				RETURN;
			END_IF

		(* Ein Link ohne Kommunikation wurde festgestellt *)
		ELSIF Q_arrDiagSlaveInfo[0].stState.bLinkError THEN

			IQ_stMeldung[nIndexErrorMessage].SourceName	:=	'EtherCAT-Bus';
			IQ_stMeldung[nIndexErrorMessage].sText :=
				CONCAT(	'Fehler EtherCAT-Bus: Teilnehmer: ',
							Q_arrDiagSlaveInfo[0].sName);

			IQ_stMeldung[nIndexErrorMessage].sText :=
				CONCAT(	IQ_stMeldung[nIndexErrorMessage].sText,
							', Typ: ');

			IQ_stMeldung[nIndexErrorMessage].sText :=
				CONCAT(	IQ_stMeldung[nIndexErrorMessage].sText,
							Q_arrDiagSlaveInfo[0].sType);

			IF Q_arrDiagSlaveInfo[0].stState.bPortA THEN
				IQ_stMeldung[nIndexErrorMessage].sText :=
						CONCAT(	IQ_stMeldung[nIndexErrorMessage].sText,
									': Am Port A wurde ein Link ohne Kommunikation festgestellt !');
			ELSIF Q_arrDiagSlaveInfo[0].stState.bPortB THEN
				IQ_stMeldung[nIndexErrorMessage].sText :=
					CONCAT(	IQ_stMeldung[nIndexErrorMessage].sText,
									': Am Port B wurde ein Link ohne Kommunikation festgestellt !');
			ELSIF Q_arrDiagSlaveInfo[0].stState.bPortC THEN
				IQ_stMeldung[nIndexErrorMessage].sText :=
					CONCAT(	IQ_stMeldung[nIndexErrorMessage].sText,
									': Am Port C wurde ein Link ohne Kommunikation festgestellt !');
			ELSIF Q_arrDiagSlaveInfo[0].stState.bPortD THEN
				IQ_stMeldung[nIndexErrorMessage].sText :=
					CONCAT(	IQ_stMeldung[nIndexErrorMessage].sText,
									': Am Port D wurde ein Link ohne Kommunikation festgestellt !');
			END_IF

			IF nIndexErrorMessage < cMaxAnzahlSlaveError THEN
				nIndexErrorMessage := nIndexErrorMessage + 1;
			ELSE
				RETURN;
			END_IF

		END_IF

	ELSE
		(* Vendor-Id, Produkt-Code, Revisions-Nummer oder Serien-Nummer des EtherCAT-Gerätes ist ungültig *)
		IF Q_arrDiagSlaveInfo[0].stState.bInvalidVPRS THEN

			IQ_stMeldung[nIndexErrorMessage].SourceName	:=	'EtherCAT-Bus';
			IQ_stMeldung[nIndexErrorMessage].sText :=
				CONCAT(	'Fehler EtherCAT-Bus: Teilnehmer: ',
							Q_arrDiagSlaveInfo[0].sName);

			IQ_stMeldung[nIndexErrorMessage].sText :=
				CONCAT(	IQ_stMeldung[nIndexErrorMessage].sText,
							', Typ: ');

			IQ_stMeldung[nIndexErrorMessage].sText :=
				CONCAT(	IQ_stMeldung[nIndexErrorMessage].sText,
							Q_arrDiagSlaveInfo[0].sType);

			IQ_stMeldung[nIndexErrorMessage].sText :=
				CONCAT(	IQ_stMeldung[nIndexErrorMessage].sText,
							'  VPRS-Fehler !');

		(* EtherCAT-Gerät ist im Status xxx *)
		ELSE

			IQ_stMeldung[nIndexErrorMessage].SourceName	:=	'EtherCAT-Bus';
			IQ_stMeldung[nIndexErrorMessage].sText :=
				CONCAT(	'Fehler EtherCAT-Bus: Teilnehmer: ',
							Q_arrDiagSlaveInfo[0].sName);

			IQ_stMeldung[nIndexErrorMessage].sText :=
				CONCAT(	IQ_stMeldung[nIndexErrorMessage].sText,
							', Typ: ');

			IQ_stMeldung[nIndexErrorMessage].sText :=
				CONCAT(	IQ_stMeldung[nIndexErrorMessage].sText,
							Q_arrDiagSlaveInfo[0].sType);

			IQ_stMeldung[nIndexErrorMessage].sText :=
				CONCAT(	IQ_stMeldung[nIndexErrorMessage].sText,
							': State: ');

			CASE Q_arrDiagSlaveInfo[0].stState.eEcState OF
	
			eEcState_UNDEFINED:	IQ_stMeldung[nIndexErrorMessage].sText :=
											CONCAT(	IQ_stMeldung[nIndexErrorMessage].sText,
														'UNDEFINED');
			eEcState_INIT:			IQ_stMeldung[nIndexErrorMessage].sText :=
											CONCAT(	IQ_stMeldung[nIndexErrorMessage].sText,
														'INIT / NO_COMMUNICATION');
			eEcState_PREOP:		IQ_stMeldung[nIndexErrorMessage].sText :=
											CONCAT(	IQ_stMeldung[nIndexErrorMessage].sText,
														'PREOP');
			eEcState_BOOT:			IQ_stMeldung[nIndexErrorMessage].sText :=
											CONCAT(	IQ_stMeldung[nIndexErrorMessage].sText,
														'BOOT');
			eEcState_SAFEOP:		IQ_stMeldung[nIndexErrorMessage].sText :=
											CONCAT(	IQ_stMeldung[nIndexErrorMessage].sText,
														'SAFEOP');
			eEcState_OP:			IQ_stMeldung[nIndexErrorMessage].sText :=
											CONCAT(	IQ_stMeldung[nIndexErrorMessage].sText,
														'OP');
			END_CASE

		END_IF

		IF nIndexErrorMessage < cMaxAnzahlSlaveError THEN
			nIndexErrorMessage := nIndexErrorMessage + 1;
		ELSE
			RETURN;
		END_IF

		(* --- *)

		(* Vendor-Id, Produkt-Code, Revisions-Nummer oder Serien-Nummer des EtherCAT-Gerätes ist ungültig *)
		IF Q_arrDiagSlaveInfo[0].stState.bInvalidVPRS THEN

			IQ_stMeldung[nIndexErrorMessage].SourceName	:=	'EtherCAT-Bus';
			IQ_stMeldung[nIndexErrorMessage].sText :=
				CONCAT(	'Fehler Teilnehmer: ',
							Q_arrDiagSlaveInfo[0].sName);

			IQ_stMeldung[nIndexErrorMessage].sText :=
				CONCAT(	IQ_stMeldung[nIndexErrorMessage].sText,
							': Konfigurierter Typ: ');

			IQ_stMeldung[nIndexErrorMessage].sText :=
				CONCAT(	IQ_stMeldung[nIndexErrorMessage].sText,
								Q_arrDiagSlaveInfo[0].sType);

			IQ_stMeldung[nIndexErrorMessage].sText :=
				CONCAT(	IQ_stMeldung[nIndexErrorMessage].sText,
							', Erkannter Typ: ');

			IQ_stMeldung[nIndexErrorMessage].sText :=
				CONCAT(	IQ_stMeldung[nIndexErrorMessage].sText,
								Q_arrDiagSlaveInfoScanned[0].sType);

			IF nIndexErrorMessage < cMaxAnzahlSlaveError THEN
				nIndexErrorMessage := nIndexErrorMessage + 1;
			ELSE
				RETURN;
			END_IF
		END_IF

	END_CASE

	(* --------------------------------------------------------------------------------------- *)
	nIndexSlave := 1;
	IF Q_arrDiagSlaveInfo[nIndexSlave].bDiagData THEN
		k_SlaveErrorMessage();
	END_IF

	(* --------------------------------------------------------------------------------------- *)
	nIndexSlave := 2;
	IF Q_arrDiagSlaveInfo[nIndexSlave].bDiagData THEN
		k_SlaveErrorMessage();
	END_IF

	(* --------------------------------------------------------------------------------------- *)
	nIndexSlave := 3;
	IF Q_arrDiagSlaveInfo[nIndexSlave].bDiagData THEN
		k_SlaveErrorMessage();
	END_IF

	(* --------------------------------------------------------------------------------------- *)

END_IF

// ENDE
END_ACTION

ACTION j_CheckMasterDevState:
//*****************************************************************************
// check master errors based on devstate
Q_bMasterDevStateError 					:=
	I_nMasterDevState <> 0;

Q_stMasterDevState.bLinkError 			:=
	((I_nMasterDevState
		AND 16#000F) = 1)
	OR((I_nMasterDevState
		AND 16#000F) = 4);

Q_stMasterDevState.bResetRequired 		:=
	((I_nMasterDevState
		AND 16#000F) = 2)
	OR((I_nMasterDevState
		AND 16#FFF0) = 16#10);

Q_stMasterDevState.bMissFrmRedMode 	:=
	(I_nMasterDevState
		AND 16#000F) = 8;

Q_stMasterDevState.bWatchdogTriggerd 	:=
	(I_nMasterDevState
		AND 16#20) = 16#20;

Q_stMasterDevState.bDriverNotFound 	:=
	(I_nMasterDevState
		AND 16#40) = 16#40;

Q_stMasterDevState.bResetActive 		:=
	(I_nMasterDevState
		AND 16#80) = 16#80;

Q_stMasterDevState.bAtLeastOneNotInOp :=
	((I_nMasterDevState
		AND 16#100) = 16#100)
	OR ((I_nMasterDevState
		AND 16#200) = 16#200)
	OR((I_nMasterDevState
		AND 16#400) = 16#400)
	OR ((I_nMasterDevState
		AND 16#800) = 16#800);

